// TwinCAT 3 PLC project ServerSampleProject
// ProgramVersion: 3.1.4026.23
// libraries:
//   Tc2_Standard, * (Beckhoff Automation GmbH)
//   Tc2_System, * (Beckhoff Automation GmbH)
//   Tc3_EventLogger, * (Beckhoff Automation GmbH)
//   Tc3_Module, * (Beckhoff Automation GmbH)
// project tree:
//   DUTs/Enums/ E_Enum_2.TcDUT, E_Operation.TcDUT, E_Enum_1.TcDUT
//   DUTs/Structures/ ST_Complex_1.TcDUT, ST_Complex_3.TcDUT, ST_Complex_4.TcDUT, ST_Complex_5.TcDUT, ST_Complex_6.TcDUT, ST_Complex_7.TcDUT, ST_Complex_8.TcDUT, ST_MathematicResults.TcDUT, ST_MathOperation.TcDUT, ST_Complex_2.TcDUT
//   GVLs/ GVL_alarm_condition.TcGVL, GVL_analog_items.TcGVL, GVL_historizing.TcGVL, GVL_inheritance.TcGVL, GVL_properties.TcGVL, Settings.TcGVL, GVL_enums.TcGVL, GVL_methods.TcGVL, GVL_structures.TcGVL, GVL_nodes_dynamic.TcGVL, GVL_nodes_static.TcGVL
//   / PlcTask.TcTTO
//   POUs/Inheritance/ FB_Base.TcPOU, FB_Derived.TcPOU
//   POUs/ MAIN.TcPOU
//   POUs/Methods/ FB_Job.TcPOU, FB_Mathematics.TcPOU, FB_Methods.TcPOU
//   POUs/Programs/ PRG_AlarmsConditions.TcPOU, PRG_Dynamic.TcPOU, PRG_Eventlogger.TcPOU, PRG_HistoricalAccess.TcPOU, PRG_Methods.TcPOU, PRG_Static.TcPOU
//   POUs/Properties/ FB_Properties.TcPOU
// real-time tasks:
//   TASK PlcTask: cycle T#10ms, priority 20, ADS port 350

CONFIGURATION ServerSampleProject
    RESOURCE PLC ON TwinCAT3
        TASK PlcTask(INTERVAL := T#10ms, PRIORITY := 20);
        PROGRAM MAIN WITH PlcTask : MAIN;
    END_RESOURCE
END_CONFIGURATION

// ---- DUTs/Enums/E_Enum_2.TcDUT
TYPE E_Enum_2 :
(
	ZERO := 0,
	ONE := 1,
	TWO := 2,
	THREE := 3,
	THIRTEEN := 13,
	the_answer_to_life_the_universe_and_everything := 42
) INT;
END_TYPE

// ---- DUTs/Enums/E_Operation.TcDUT
TYPE E_Operation :
(
	Addition := 0,
	Substract,
	Multiply,
	Divide
);
END_TYPE

// ---- DUTs/Enums/E_Enum_1.TcDUT
TYPE E_Enum_1 :
(
	ZERO := 0,
	ONE := 1,
	TWO := 2,
	THREE := 3,
	THIRTEEN := 13,
	the_answer_to_life_the_universe_and_everything := 42
);
END_TYPE

// ---- DUTs/Structures/ST_Complex_1.TcDUT
{attribute 'OPC.UA.DA' := '1'}
{attribute 'OPC.UA.DA.StructuredType' := '1'}
TYPE ST_Complex_1 :
STRUCT
	x 	: E_Enum_1;
	a 	: DINT;
	str : STRING;
	b 	: DINT;
END_STRUCT
END_TYPE

// ---- DUTs/Structures/ST_Complex_3.TcDUT
{attribute 'OPC.UA.DA' := '1'}
{attribute 'OPC.UA.DA.StructuredType' := '1'}
TYPE ST_Complex_3 :
STRUCT
	stAmsAddr : ST_AmsAddr;
END_STRUCT
END_TYPE

// ---- DUTs/Structures/ST_Complex_4.TcDUT
{attribute 'OPC.UA.DA' := '1'}
{attribute 'OPC.UA.DA.StructuredType' := '1'}
TYPE ST_Complex_4 :
STRUCT
	ErrorID : E_Enum_1;
END_STRUCT
END_TYPE

// ---- DUTs/Structures/ST_Complex_5.TcDUT
TYPE ST_Complex_5 :
STRUCT
	a : INT := 42;
	b : DINT := 43;
	c : REAL := 42.42;
	d : LREAL := 42.42;
	e : STRING := 'Hello TwinCAT';
	f : INT := 42;
	g : BOOL := TRUE;
END_STRUCT
END_TYPE

// ---- DUTs/Structures/ST_Complex_6.TcDUT
TYPE ST_Complex_6 :
STRUCT
	a : INT := 42;
	b : DINT := 43;
	c : REAL := 42.42;
	d : LREAL := 42.42;
	e : INT := 44;
	f : BOOL := TRUE;
END_STRUCT
END_TYPE

// ---- DUTs/Structures/ST_Complex_7.TcDUT
TYPE ST_Complex_7 :
STRUCT
	a : LREAL := 42.42;
	b : REAL := 42.42;
	c : REAL := 42.42;
END_STRUCT
END_TYPE

// ---- DUTs/Structures/ST_Complex_8.TcDUT
{attribute 'OPC.UA.DA' := '1'}
{attribute 'OPC.UA.DA.StructuredType' := '1'}
TYPE ST_Complex_8 :
STRUCT
	stComplex		: ST_Complex_1;
	strString5		: STRING[5]; (*String, max 5 chars*)
	eEnum	 		: E_Enum_1;
	strString3	 	: STRING[3]; (*String, max 3 chars*)
	arrComplex 		: ARRAY[0..1] OF ST_Complex_1;
	arrDint		 	: ARRAY[0..100] OF DINT;	
END_STRUCT
END_TYPE

// ---- DUTs/Structures/ST_MathematicResults.TcDUT
TYPE ST_MathematicResults :
STRUCT
	Sum : LREAL;
	Diff : LREAL;
	Prod : LREAL;
	Quo : LREAL;
END_STRUCT
END_TYPE

// ---- DUTs/Structures/ST_MathOperation.TcDUT
{attribute 'OPC.UA.DA.Description' := 'Structure to describe a math operation having one operator and two oparands'}
TYPE ST_MathOperation :
STRUCT
	operator : E_OPERATION; (*define the operator for calculation*)
	a : LREAL; (*First operand*)
	b : LREAL; (*Second operand*)
END_STRUCT
END_TYPE

// ---- DUTs/Structures/ST_Complex_2.TcDUT
{attribute 'OPC.UA.DA' := '1'}
{attribute 'OPC.UA.DA.StructuredType' := '1'}
TYPE ST_Complex_2 :
STRUCT
	c1 		: ST_Complex_1;
	s_5 	: STRING[5]; (*String, max 5 chars*)
	e 		: E_Enum_1;
	s_3 	: STRING[3]; (*String, max 3 chars*)
	cArr 	: ARRAY[0..5] OF ST_Complex_1;
	iArr 	: ARRAY[0..100] OF DINT;	
END_STRUCT
END_TYPE

// ---- GVLs/GVL_alarm_condition.TcGVL
VAR_GLOBAL
	{attribute 'OPC.UA.DA' := '1'}
	{attribute 'OPC.UA.DA.Description' := 'Triggers a LimitAlarmType when value reaches 10 or 0. Increments every 10 secs'}
	limitAlmTrigger: DINT;
	
	{attribute 'OPC.UA.DA' := '1'}
	{attribute 'OPC.UA.DA.Description' := 'Triggers an OffNormalAlarmType when set to true. State changes state every 10 secs.'}
	offNormAlmTrigger : BOOL;
END_VAR

// ---- GVLs/GVL_analog_items.TcGVL
{attribute 'qualified_only'}
VAR_GLOBAL
	{attribute 'OPC.UA.DA' := '1'}
	{attribute 'OPC.UA.DA.AnalogItemType' := '1'}
	{attribute 'OPC.UA.DA.AnalogItemType.EngineeringUnits' := '20529'  }(*EngeneeringUnit = percent*)
	{attribute 'OPC.UA.DA.AnalogItemType.InstrumentRange' := '0:100'  }
	{attribute 'OPC.UA.DA.AnalogItemType.EURange' := '10:90'  }
	{attribute 'OPC.UA.DA.AnalogItemType.WriteBehavior' := '1'  } (*AnalogWrMode_AllowAny = 0,
																	AnalogWrMode_Clamp = 1,
																	AnalogWrMode_Reject = 2,*)
	{attribute 'OPC.UA.DA.Description' := 'Analog item type. Write mode is clamped to instrument range'}
	analog_percent : REAL := 50;
	
	{attribute 'OPC.UA.DA' := '1'}
	{attribute 'OPC.UA.DA.AnalogItemType' := '1'}
	{attribute 'OPC.UA.DA.AnalogItemType.EngineeringUnits' := '12851'  }(*EngeneeringUnit = gram_per_cubic_centimetre*)
	{attribute 'OPC.UA.DA.AnalogItemType.InstrumentRange' := '0:100'  }
	{attribute 'OPC.UA.DA.AnalogItemType.EURange' := '0:75'  }
	{attribute 'OPC.UA.DA.AnalogItemType.WriteBehavior' := '2'  } (*AnalogWrMode_AllowAny = 0,
																	AnalogWrMode_Clamp = 1,
																	AnalogWrMode_Reject = 2,*)
	{attribute 'OPC.UA.DA.Description' := 'Analog item type. Write is rejected when out of instrument range'}
	analog_gram_per_cubic_centimetre : REAL := 50;	
	
	{attribute 'OPC.UA.DA' := '1'}
	{attribute 'OPC.UA.DA.AnalogItemType' := '1'}
	{attribute 'OPC.UA.DA.AnalogItemType.EngineeringUnits' := '5257525'  }(*EngeneeringUnit = megabyte_per_second*)
	{attribute 'OPC.UA.DA.AnalogItemType.EURange' := '0:10'  }
	{attribute 'OPC.UA.DA.AnalogItemType.InstrumentRange' := '0:100'  }
	{attribute 'OPC.UA.DA.AnalogItemType.WriteBehavior' := '0'  } (*AnalogWrMode_AllowAny = 0,
																	AnalogWrMode_Clamp = 1,
																	AnalogWrMode_Reject = 2,*)
	{attribute 'OPC.UA.DA.Description' := 'Analog item type. Write mode allows writing out of Instrument range'}
	analog_mbps : REAL;	
	
	{attribute 'OPC.UA.DA' := '1'}
	{attribute 'OPC.UA.DA.AnalogItemType' := '1'}
	{attribute 'OPC.UA.DA.AnalogItemType.EngineeringUnits' := '20529'  }(*EngeneeringUnit = percent*)
	{attribute 'OPC.UA.DA.AnalogItemType.InstrumentRange' := '0:100'  }
	{attribute 'OPC.UA.DA.AnalogItemType.EURange' := '10:90'  }
	{attribute 'OPC.UA.DA.AnalogItemType.WriteBehavior' := '2'  } (*AnalogWrMode_AllowAny = 0,
																	AnalogWrMode_Clamp = 1,
																	AnalogWrMode_Reject = 2,*)
	{attribute 'OPC.UA.DA.Description' := 'Analog item of type Double. '}
	analog_dbl : LREAL := 50;	
	
	{attribute 'OPC.UA.DA' := '1'}
	{attribute 'OPC.UA.DA.AnalogItemType' := '1'}
	{attribute 'OPC.UA.DA.AnalogItemType.EngineeringUnits' := '20529'  }(*EngeneeringUnit = percent*)
	{attribute 'OPC.UA.DA.AnalogItemType.InstrumentRange' := '0:100'  }
	{attribute 'OPC.UA.DA.AnalogItemType.EURange' := '10:90'  }
	{attribute 'OPC.UA.DA.AnalogItemType.WriteBehavior' := '2'  } (*AnalogWrMode_AllowAny = 0,
																	AnalogWrMode_Clamp = 1,
																	AnalogWrMode_Reject = 2,*)
	{attribute 'OPC.UA.DA.Description' := 'Analog item of type Float. '}
	analog_flt : REAL := 50;		
	
	{attribute 'OPC.UA.DA' := '1'}
	{attribute 'OPC.UA.DA.AnalogItemType' := '1'}
	{attribute 'OPC.UA.DA.AnalogItemType.EngineeringUnits' := '20529'  }(*EngeneeringUnit = percent*)
	{attribute 'OPC.UA.DA.AnalogItemType.InstrumentRange' := '0:100'  }
	{attribute 'OPC.UA.DA.AnalogItemType.EURange' := '10:90'  }
	{attribute 'OPC.UA.DA.AnalogItemType.WriteBehavior' := '2'  } (*AnalogWrMode_AllowAny = 0,
																	AnalogWrMode_Clamp = 1,
																	AnalogWrMode_Reject = 2,*)
	{attribute 'OPC.UA.DA.Description' := 'Analog item of type Int16. '}
	analog_i16 : INT := 50;		
	
	{attribute 'OPC.UA.DA' := '1'}
	{attribute 'OPC.UA.DA.AnalogItemType' := '1'}
	{attribute 'OPC.UA.DA.AnalogItemType.EngineeringUnits' := '20529'  }(*EngeneeringUnit = percent*)
	{attribute 'OPC.UA.DA.AnalogItemType.InstrumentRange' := '0:100'  }
	{attribute 'OPC.UA.DA.AnalogItemType.EURange' := '10:90'  }
	{attribute 'OPC.UA.DA.AnalogItemType.WriteBehavior' := '2'  } (*AnalogWrMode_AllowAny = 0,
																	AnalogWrMode_Clamp = 1,
																	AnalogWrMode_Reject = 2,*)
	{attribute 'OPC.UA.DA.Description' := 'Analog item of type UInt16. '}
	analog_ui16 : UINT := 50;		
	
	{attribute 'OPC.UA.DA' := '1'}
	{attribute 'OPC.UA.DA.AnalogItemType' := '1'}
	{attribute 'OPC.UA.DA.AnalogItemType.EngineeringUnits' := '20529'  }(*EngeneeringUnit = percent*)
	{attribute 'OPC.UA.DA.AnalogItemType.InstrumentRange' := '0:100'  }
	{attribute 'OPC.UA.DA.AnalogItemType.EURange' := '10:90'  }
	{attribute 'OPC.UA.DA.AnalogItemType.WriteBehavior' := '2'  } (*AnalogWrMode_AllowAny = 0,
																	AnalogWrMode_Clamp = 1,
																	AnalogWrMode_Reject = 2,*)
	{attribute 'OPC.UA.DA.Description' := 'Analog item of type Int32. '}
	analog_i32 : DINT := 50;		

	{attribute 'OPC.UA.DA' := '1'}
	{attribute 'OPC.UA.DA.AnalogItemType' := '1'}
	{attribute 'OPC.UA.DA.AnalogItemType.EngineeringUnits' := '20529'  }(*EngeneeringUnit = percent*)
	{attribute 'OPC.UA.DA.AnalogItemType.InstrumentRange' := '0:100'  }
	{attribute 'OPC.UA.DA.AnalogItemType.EURange' := '10:90'  }
	{attribute 'OPC.UA.DA.AnalogItemType.WriteBehavior' := '2'  } (*AnalogWrMode_AllowAny = 0,
																	AnalogWrMode_Clamp = 1,
																	AnalogWrMode_Reject = 2,*)
	{attribute 'OPC.UA.DA.Description' := 'Analog item of type UInt32. '}
	analog_ui32 : UDINT := 50;
	
	{attribute 'OPC.UA.DA' := '1'}
	{attribute 'OPC.UA.DA.AnalogItemType' := '1'}
	{attribute 'OPC.UA.DA.AnalogItemType.EngineeringUnits' := '20529'  }(*EngeneeringUnit = percent*)
	{attribute 'OPC.UA.DA.AnalogItemType.InstrumentRange' := '0:100'  }
	{attribute 'OPC.UA.DA.AnalogItemType.EURange' := '10:90'  }
	{attribute 'OPC.UA.DA.AnalogItemType.WriteBehavior' := '2'  } (*AnalogWrMode_AllowAny = 0,
																	AnalogWrMode_Clamp = 1,
																	AnalogWrMode_Reject = 2,*)
	{attribute 'OPC.UA.DA.Description' := 'Analog item of type Int64. '}
	analog_i64 : LINT := 50;		
	
	{attribute 'OPC.UA.DA' := '1'}
	{attribute 'OPC.UA.DA.AnalogItemType' := '1'}
	{attribute 'OPC.UA.DA.AnalogItemType.EngineeringUnits' := '20529'  }(*EngeneeringUnit = percent*)
	{attribute 'OPC.UA.DA.AnalogItemType.InstrumentRange' := '0:100'  }
	{attribute 'OPC.UA.DA.AnalogItemType.EURange' := '10:90'  }
	{attribute 'OPC.UA.DA.AnalogItemType.WriteBehavior' := '2'  } (*AnalogWrMode_AllowAny = 0,
																	AnalogWrMode_Clamp = 1,
																	AnalogWrMode_Reject = 2,*)
	{attribute 'OPC.UA.DA.Description' := 'Analog item of type UInt64. '}
	analog_ui64 : ULINT := 50;		
	
	{attribute 'OPC.UA.DA' := '1'}
	{attribute 'OPC.UA.DA.AnalogItemType' := '1'}
	{attribute 'OPC.UA.DA.AnalogItemType.EngineeringUnits' := '20529'  }(*EngeneeringUnit = percent*)
	{attribute 'OPC.UA.DA.AnalogItemType.InstrumentRange' := '0:100'  }
	{attribute 'OPC.UA.DA.AnalogItemType.EURange' := '10:90'  }
	{attribute 'OPC.UA.DA.AnalogItemType.WriteBehavior' := '2'  } (*AnalogWrMode_AllowAny = 0,
																	AnalogWrMode_Clamp = 1,
																	AnalogWrMode_Reject = 2,*)
	{attribute 'OPC.UA.DA.Description' := 'Analog item of type SByte. '}
	analog_i8 : SINT := 50;		
	
	{attribute 'OPC.UA.DA' := '1'}
	{attribute 'OPC.UA.DA.AnalogItemType' := '1'}
	{attribute 'OPC.UA.DA.AnalogItemType.EngineeringUnits' := '20529'  }(*EngeneeringUnit = percent*)
	{attribute 'OPC.UA.DA.AnalogItemType.InstrumentRange' := '0:100'  }
	{attribute 'OPC.UA.DA.AnalogItemType.EURange' := '10:90'  }
	{attribute 'OPC.UA.DA.AnalogItemType.WriteBehavior' := '2'  } (*AnalogWrMode_AllowAny = 0,
																	AnalogWrMode_Clamp = 1,
																	AnalogWrMode_Reject = 2,*)
	{attribute 'OPC.UA.DA.Description' := 'Analog item of type Byte. '}
	analog_ui8 : USINT := 50;	
END_VAR

// ---- GVLs/GVL_historizing.TcGVL
VAR_GLOBAL
	
	{attribute 'OPC.UA.DA' := '1'}
	{attribute 'OPC.UA.DA.Description' := 'HistoricalAccess with Volatile storage'}
	volatile_sinus	: LREAL;
	{attribute 'OPC.UA.DA' := '1'}
	{attribute 'OPC.UA.DA.Description' := 'HistoricalAccess with Volatile storage'}	
	volatile_cosinus : LREAL;
	{attribute 'OPC.UA.DA' := '1'}
	{attribute 'OPC.UA.DA.Description' := 'HistoricalAccess with Volatile storage'}	
	volatile_cosinushalf : LREAL;
	{attribute 'OPC.UA.DA' := '1'}
	{attribute 'OPC.UA.DA.Description' := 'HistoricalAccess with SQLite storage'}
	sqlite_sinus : LREAL;
	{attribute 'OPC.UA.DA' := '1'}
	{attribute 'OPC.UA.DA.Description' := 'HistoricalAccess with SQLite storage'}	
	sqlite_cosinus : LREAL;
	{attribute 'OPC.UA.DA' := '1'}
	{attribute 'OPC.UA.DA.Description' := 'HistoricalAccess with SQLite storage'}	
	sqlite_cosinushalf : LREAL;

END_VAR

// ---- GVLs/GVL_inheritance.TcGVL
{attribute 'qualified_only'}
VAR_GLOBAL
	{attribute 'OPC.UA.DA' := '1'}
	{attribute 'OPC.UA.DA.Description' := 'Base class'}
	BaseType : FB_Base;
	
	{attribute 'OPC.UA.DA' := '1'}
	{attribute 'OPC.UA.DA.Description' := 'Derived class'}
	DerivedType : FB_Derived;	
END_VAR

// ---- GVLs/GVL_properties.TcGVL
{attribute 'qualified_only'}
VAR_GLOBAL
	{attribute 'OPC.UA.DA' := '1'}
	Properties : FB_Properties;
END_VAR

// ---- GVLs/Settings.TcGVL
VAR_GLOBAL
	{attribute 'OPC.UA.DA' := '1'}
	{attribute 'OPC.UA.DA.Description' := 'Sets PLC update interval of variables in GVL_nodes_dynamic'} 	
	UpdateTimer : TON := (PT:=T#10MS);
END_VAR
VAR_GLOBAL CONSTANT
	ARRSIZEX : INT := 10; 
	ARRSIZEY : INT := 10; 
	ARRSIZEZ : INT := 10;
	ARRSIZEHUGE : INT := 10000;
END_VAR

// ---- GVLs/GVL_enums.TcGVL
{attribute 'qualified_only'}
VAR_GLOBAL
	{attribute 'OPC.UA.DA' := '1'}
	{attribute 'OPC.UA.DA.Description' := 'Enumeration type (DINT)'} 
	Enum1 : E_Enum_1;
	{attribute 'OPC.UA.DA' := '1'}
	{attribute 'OPC.UA.DA.Description' := 'Enumeration type (INT)'} 
	Enum2 : E_Enum_2;	
END_VAR

// ---- GVLs/GVL_methods.TcGVL
VAR_GLOBAL
	{attribute 'OPC.UA.DA' := '1'}
	{attribute 'OPC.UA.DA.Description' := 'Methods with different InputOutput types'} 	
	Methods : FB_Methods;
	
	{attribute 'OPC.UA.DA' := '1'}
	{attribute 'OPC.UA.DA.Description' := 'Methods with mathematical functions'}
	Mathematics : FB_Mathematics;

	{attribute 'OPC.UA.DA' := '1'}
	{attribute 'OPC.UA.DA.Description' := 'Job method which execution may take longer than a PLC cycle'}
	Job : FB_Job;	
END_VAR

// ---- GVLs/GVL_structures.TcGVL
VAR_GLOBAL
	{attribute 'OPC.UA.DA' := '1'}
	{attribute 'OPC.UA.DA.StructuredType' := '1'}
	{attribute 'OPC.UA.DA.Description' := 'Complex (structured) type '} 	
	StructuredType1 : ST_Complex_1;
	
	{attribute 'OPC.UA.DA' := '2'}
	{attribute 'OPC.UA.DA.StructuredType' := '1'}
	{attribute 'OPC.UA.DA.Description' := 'Complex (structured) type '} 	
	StructuredType1WithoutMember : ST_Complex_1;

	{attribute 'OPC.UA.DA' := '1'}
	{attribute 'OPC.UA.DA.StructuredType' := '1'}
	{attribute 'OPC.UA.DA.Description' := 'Complex (structured) type '} 		
	StructuredType2 : ST_Complex_2;
	
	{attribute 'OPC.UA.DA' := '1'}
	{attribute 'OPC.UA.DA.StructuredType' := '1'}
	{attribute 'OPC.UA.DA.Description' := 'Complex (structured) type '} 		
	StructuredType3 : ST_Complex_3;

	{attribute 'OPC.UA.DA' := '1'}
	{attribute 'OPC.UA.DA.StructuredType' := '1'}
	{attribute 'OPC.UA.DA.Description' := 'Complex (structured) type '} 		
	StructuredType4 : ST_Complex_4;	
	
	{attribute 'OPC.UA.DA' := '1'}
	{attribute 'OPC.UA.DA.StructuredType' := '1'}
	{attribute 'OPC.UA.DA.Description' := 'Complex (structured) type '} 		
	StructuredType5 : ST_Complex_5;	
	
	{attribute 'OPC.UA.DA' := '1'}
	{attribute 'OPC.UA.DA.StructuredType' := '1'}
	{attribute 'OPC.UA.DA.Description' := 'Complex (structured) type '} 		
	StructuredType6 : ST_Complex_6;	
	
	{attribute 'OPC.UA.DA' := '1'}
	{attribute 'OPC.UA.DA.StructuredType' := '1'}
	{attribute 'OPC.UA.DA.Description' := 'Complex (structured) type '} 		
	StructuredType7 : ST_Complex_7;		

	{attribute 'OPC.UA.DA' := '1'}
	{attribute 'OPC.UA.DA.StructuredType' := '1'}
	{attribute 'OPC.UA.DA.Description' := 'Complex (structured) type '} 		
	StructuredType8 : ST_Complex_8;	
	
	{attribute 'OPC.UA.DA' := '1'}
	{attribute 'OPC.UA.DA.StructuredType' := '1'}
	{attribute 'OPC.UA.DA.Description' := 'Array of complex (structured) type'} 	
	arrStComplex : ARRAY[0..ARRSIZEX] OF ST_Complex_1;

	{attribute 'OPC.UA.DA' := '1'}
	{attribute 'OPC.UA.DA.StructuredType' := '1'}
	{attribute 'OPC.UA.DA.Description' := 'Array of complex (structured) type'} 		
	arrStComplex2 : ARRAY[0..ARRSIZEX] OF ST_Complex_2;		
END_VAR

// ---- GVLs/GVL_nodes_dynamic.TcGVL
VAR_GLOBAL
	//scalars
	{attribute 'OPC.UA.DA' := '1'}
	{attribute 'OPC.UA.DA.Description' := 'Scalar BOOL, modified by a TRIG'}	
	dyn_scalar_BOOL_trigger : BOOL;
	{attribute 'OPC.UA.DA' := '1'}
	{attribute 'OPC.UA.DA.Description' := 'Scalar BOOL'} 
	dyn_scalar_BOOL	: BOOL;(* ~ 	(OPC : 1 : available for OPC-clients) *)
	{attribute 'OPC.UA.DA' := '1'}
	{attribute 'OPC.UA.DA.Description' := 'Scalar SINT'}
	dyn_scalar_I1	: SINT;		(* ~ 	(OPC : 1 : available for OPC-clients) *)					
	{attribute 'OPC.UA.DA' := '1'}
	{attribute 'OPC.UA.DA.Description' := 'Scalar USINT'}	
	dyn_scalar_UI1	: USINT;	(* ~ 	(OPC : 1 : available for OPC-clients) *)					
	{attribute 'OPC.UA.DA' := '1'}
	{attribute 'OPC.UA.DA.Description' := 'Scalar INT'}	
	dyn_scalar_I2 	: INT;			(* ~ 	(OPC : 1 : available for OPC-clients) *)				
	{attribute 'OPC.UA.DA' := '1'}
	{attribute 'OPC.UA.DA.Description' := 'Scalar UINT'}	
	dyn_scalar_UI2	: UINT;			(* ~ 	(OPC : 1 : available for OPC-clients) *)				
	{attribute 'OPC.UA.DA' := '1'}
	{attribute 'OPC.UA.DA.Description' := 'Scalar DINT'}	
	dyn_scalar_I4	: DINT;		(* ~ 	(OPC : 1 : available for OPC-clients) *)					
	{attribute 'OPC.UA.DA' := '1'}
	{attribute 'OPC.UA.DA.Description' := 'Scalar UDINT'}	
	dyn_scalar_UI4	: UDINT;(* ~ 	(OPC : 1 : available for OPC-clients) *)
	{attribute 'OPC.UA.DA' := '1'}
	{attribute 'OPC.UA.DA.Description' := 'Scalar LINT'}
	dyn_scalar_I8	: LINT;	(* ~ 	(OPC : 1 : available for OPC-clients) *)
	{attribute 'OPC.UA.DA' := '1'}
	{attribute 'OPC.UA.DA.Description' := 'Scalar ULINT'}
	dyn_scalar_UI8	: ULINT;(* ~ 	(OPC : 1 : available for OPC-clients) *)
	{attribute 'OPC.UA.DA' := '1'}
	{attribute 'OPC.UA.DA.Description' := 'Scalar BYTE'}
	dyn_scalar_BYTE	: BYTE;(* ~ 	(OPC : 1 : available for OPC-clients) *)
	{attribute 'OPC.UA.DA' := '1'}
	{attribute 'OPC.UA.DA.Description' := 'Scalar WORD'}	
	dyn_scalar_WORD	: WORD;(* ~ 	(OPC : 1 : available for OPC-clients) *)
	{attribute 'OPC.UA.DA' := '1'}
	{attribute 'OPC.UA.DA.Description' := 'Scalar DWORD'}	
	dyn_scalar_DWORD: DWORD;(* ~ 	(OPC : 1 : available for OPC-clients) *)
	{attribute 'OPC.UA.DA' := '1'}
	{attribute 'OPC.UA.DA.Description' := 'Scalar LWORD'}	
	dyn_scalar_LWORD: LWORD;(* ~ 	(OPC : 1 : available for OPC-clients) *)
	{attribute 'OPC.UA.DA' := '1'}
	{attribute 'OPC.UA.DA.Description' := 'Scalar REAL'}	
	dyn_scalar_R4	: REAL;(* ~ 	(OPC : 1 : available for OPC-clients) *)
	{attribute 'OPC.UA.DA' := '1'}
	{attribute 'OPC.UA.DA.Description' := 'Scalar LREAL'}
	dyn_scalar_R8	: LREAL;(* ~ 	(OPC : 1 : available for OPC-clients) *)
	{attribute 'OPC.UA.DA' := '1'}
	{attribute 'OPC.UA.DA.Description' := 'Scalar STRING'}	
	dyn_scalar_BSTR	: STRING;(* ~ 	(OPC : 1 : available for OPC-clients) *)
	{attribute 'OPC.UA.DA' := '1'}
	{attribute 'OPC.UA.DA.Description' := 'Scalar CHAR'}	
	//dyn_scalar_CHAR	: CHAR;
	{attribute 'OPC.UA.DA' := '1'}
	{attribute 'OPC.UA.DA.Description' := 'Scalar WSTRING'}	
	dyn_scalar_WSTRING : WSTRING;(* ~ 	(OPC : 1 : available for OPC-clients) *)
	{attribute 'OPC.UA.DA' := '1'}
	{attribute 'OPC.UA.DA.Description' := 'Scalar WCHAR'}	
	//dyn_scalar_WCHAR: WCHAR;
	{attribute 'OPC.UA.DA' := '1'}
	{attribute 'OPC.UA.DA.Description' := 'Scalar DT'}	
	dyn_scalar_DT	: DT;(* ~ 	(OPC : 1 : available for OPC-clients) *)
	{attribute 'OPC.UA.DA' := '1'}
	{attribute 'OPC.UA.DA.Description' := 'Scalar DATE'}	
	dyn_scalar_DATE : DATE;(* ~ 	(OPC : 1 : available for OPC-clients) *)
	{attribute 'OPC.UA.DA' := '1'}
	{attribute 'OPC.UA.DA.Description' := 'Scalar TOD'}	
	dyn_scalar_TOD	: TOD;(* ~ 	(OPC : 1 : available for OPC-clients) *)
	{attribute 'OPC.UA.DA' := '1'}
	{attribute 'OPC.UA.DA.Description' := 'Scalar TIME'}	
	dyn_scalar_TIME	: TIME;(* ~ 	(OPC : 1 : available for OPC-clients) *)
	
	//1dim
	{attribute 'OPC.UA.DA' := '1'}
	{attribute 'OPC.UA.DA.Description' := '1dim Array BOOL'}	
	dyn_1dim_BOOL	: ARRAY[0..ARRSIZEX] OF BOOL;(* ~ 	(OPC : 1 : available for OPC-clients) *)
	{attribute 'OPC.UA.DA' := '1'}
	{attribute 'OPC.UA.DA.Description' := '1dim Array BOOL'}	
	dyn_1dim_I1		: ARRAY[0..ARRSIZEX] OF SINT;(* ~ 	(OPC : 1 : available for OPC-clients) *)
	{attribute 'OPC.UA.DA' := '1'}
	{attribute 'OPC.UA.DA.Description' := '1dim Array BOOL'}	
	dyn_1dim_I1_Huge: ARRAY[0..ARRSIZEHUGE] OF SINT;(* ~ 	(OPC : 1 : available for OPC-clients) *)	
	{attribute 'OPC.UA.DA' := '1'}
	{attribute 'OPC.UA.DA.Description' := '1dim Array BOOL'}
	dyn_1dim_UI1	: ARRAY[0..ARRSIZEX] OF USINT;(* ~ 	(OPC : 1 : available for OPC-clients) *)
	{attribute 'OPC.UA.DA' := '1'}
	{attribute 'OPC.UA.DA.Description' := '1dim Array BOOL'}
	dyn_1dim_I2 	: ARRAY[0..ARRSIZEX] OF INT;(* ~ 	(OPC : 1 : available for OPC-clients) *)
	{attribute 'OPC.UA.DA' := '1'}
	{attribute 'OPC.UA.DA.Description' := '1dim Array BOOL'}	
	dyn_1dim_UI2	: ARRAY[0..ARRSIZEX] OF UINT;(* ~ 	(OPC : 1 : available for OPC-clients) *)
	{attribute 'OPC.UA.DA' := '1'}
	{attribute 'OPC.UA.DA.Description' := '1dim Array BOOL'}	
	dyn_1dim_I4		: ARRAY[0..ARRSIZEX] OF DINT;(* ~ 	(OPC : 1 : available for OPC-clients) *)
	{attribute 'OPC.UA.DA' := '1'}
	{attribute 'OPC.UA.DA.Description' := '1dim Array BOOL'}	
	dyn_1dim_I4_Huge: ARRAY[0..ARRSIZEHUGE] OF DINT;(* ~ 	(OPC : 1 : available for OPC-clients) *)	
	{attribute 'OPC.UA.DA' := '1'}
	{attribute 'OPC.UA.DA.Description' := '1dim Array BOOL'}
	dyn_1dim_UI4	: ARRAY[0..ARRSIZEX] OF UDINT;(* ~ 	(OPC : 1 : available for OPC-clients) *)
	{attribute 'OPC.UA.DA' := '1'}
	{attribute 'OPC.UA.DA.Description' := '1dim Array BOOL'}
	dyn_1dim_I8		: ARRAY[0..ARRSIZEX] OF LINT;(* ~ 	(OPC : 1 : available for OPC-clients) *)
	{attribute 'OPC.UA.DA' := '1'}
	{attribute 'OPC.UA.DA.Description' := '1dim Array BOOL'}
	dyn_1dim_UI8	: ARRAY[0..ARRSIZEX] OF ULINT;(* ~ 	(OPC : 1 : available for OPC-clients) *)
	{attribute 'OPC.UA.DA' := '1'}
	{attribute 'OPC.UA.DA.Description' := '1dim Array BOOL'}
	dyn_1dim_BYTE	: ARRAY[0..ARRSIZEX] OF BYTE;(* ~ 	(OPC : 1 : available for OPC-clients) *)
	{attribute 'OPC.UA.DA' := '1'}
	{attribute 'OPC.UA.DA.Description' := '1dim Array BOOL'}
	dyn_1dim_WORD	: ARRAY[0..ARRSIZEX] OF WORD;(* ~ 	(OPC : 1 : available for OPC-clients) *)
	{attribute 'OPC.UA.DA' := '1'}
	{attribute 'OPC.UA.DA.Description' := '1dim Array BOOL'}
	dyn_1dim_DWORD	: ARRAY[0..ARRSIZEX] OF DWORD;(* ~ 	(OPC : 1 : available for OPC-clients) *)
	{attribute 'OPC.UA.DA' := '1'}
	{attribute 'OPC.UA.DA.Description' := '1dim Array BOOL'}
	dyn_1dim_LWORD	: ARRAY[0..ARRSIZEX] OF LWORD;(* ~ 	(OPC : 1 : available for OPC-clients) *)
	{attribute 'OPC.UA.DA' := '1'}
	{attribute 'OPC.UA.DA.Description' := '1dim Array BOOL'}
	dyn_1dim_R4		: ARRAY[0..ARRSIZEX] OF REAL;(* ~ 	(OPC : 1 : available for OPC-clients) *)
	{attribute 'OPC.UA.DA' := '1'}
	{attribute 'OPC.UA.DA.Description' := '1dim Array BOOL'}
	dyn_1dim_R8		: ARRAY[0..ARRSIZEX] OF LREAL;(* ~ 	(OPC : 1 : available for OPC-clients) *)
	{attribute 'OPC.UA.DA' := '1'}
	{attribute 'OPC.UA.DA.Description' := '1dim Array BOOL'}
	dyn_1dim_BSTR	: ARRAY[0..ARRSIZEX] OF STRING;(* ~ 	(OPC : 1 : available for OPC-clients) *)
	{attribute 'OPC.UA.DA' := '1'}
	{attribute 'OPC.UA.DA.Description' := '1dim Array BOOL'}
	//dyn_1dim_CHAR	: ARRAY[0..ARRSIZEX] OF CHAR;
	{attribute 'OPC.UA.DA' := '1'}
	{attribute 'OPC.UA.DA.Description' := '1dim Array BOOL'}
	dyn_1dim_WSTRING : ARRAY[0..ARRSIZEX] OF WSTRING;(* ~ 	(OPC : 1 : available for OPC-clients) *)
	{attribute 'OPC.UA.DA' := '1'}
	{attribute 'OPC.UA.DA.Description' := '1dim Array BOOL'}
	//dyn_1dim_WCHAR: ARRAY[0..ARRSIZEX] OF WCHAR;
	{attribute 'OPC.UA.DA' := '1'}
	{attribute 'OPC.UA.DA.Description' := '1dim Array BOOL'}
	dyn_1dim_DT		: ARRAY[0..ARRSIZEX] OF DT;(* ~ 	(OPC : 1 : available for OPC-clients) *)
	{attribute 'OPC.UA.DA' := '1'}
	{attribute 'OPC.UA.DA.Description' := '1dim Array BOOL'}
	dyn_1dim_DATE 	: ARRAY[0..ARRSIZEX] OF DATE;(* ~ 	(OPC : 1 : available for OPC-clients) *)
	{attribute 'OPC.UA.DA' := '1'}
	{attribute 'OPC.UA.DA.Description' := '1dim Array BOOL'}
	dyn_1dim_TOD	: ARRAY[0..ARRSIZEX] OF TOD;(* ~ 	(OPC : 1 : available for OPC-clients) *)
	{attribute 'OPC.UA.DA' := '1'}
	{attribute 'OPC.UA.DA.Description' := '1dim Array BOOL'}
	dyn_1dim_TIME	: ARRAY[0..ARRSIZEX] OF TIME;(* ~ 	(OPC : 1 : available for OPC-clients) *)
	
	//2dim
	{attribute 'OPC.UA.DA' := '1'}
	{attribute 'OPC.UA.DA.Description' := '2dim Array BOOL'}
	dyn_2dim_BOOL	: ARRAY[0..ARRSIZEX, 0..ARRSIZEY] OF BOOL;(* ~ 	(OPC : 1 : available for OPC-clients) *)
	{attribute 'OPC.UA.DA' := '1'}
	{attribute 'OPC.UA.DA.Description' := '2dim Array BOOL'}
	dyn_2dim_I1		: ARRAY[0..ARRSIZEX, 0..ARRSIZEY] OF SINT;(* ~ 	(OPC : 1 : available for OPC-clients) *)
	{attribute 'OPC.UA.DA' := '1'}
	{attribute 'OPC.UA.DA.Description' := '2dim Array BOOL'}
	dyn_2dim_UI1	: ARRAY[0..ARRSIZEX, 0..ARRSIZEY] OF USINT;(* ~ 	(OPC : 1 : available for OPC-clients) *)
	{attribute 'OPC.UA.DA' := '1'}
	{attribute 'OPC.UA.DA.Description' := '2dim Array BOOL'}
	dyn_2dim_I2 	: ARRAY[0..ARRSIZEX, 0..ARRSIZEY] OF INT;(* ~ 	(OPC : 1 : available for OPC-clients) *)
	{attribute 'OPC.UA.DA' := '1'}
	{attribute 'OPC.UA.DA.Description' := '2dim Array BOOL'}
	dyn_2dim_UI2	: ARRAY[0..ARRSIZEX, 0..ARRSIZEY] OF UINT;(* ~ 	(OPC : 1 : available for OPC-clients) *)
	{attribute 'OPC.UA.DA' := '1'}
	{attribute 'OPC.UA.DA.Description' := '2dim Array BOOL'}
	dyn_2dim_I4		: ARRAY[0..ARRSIZEX, 0..ARRSIZEY] OF DINT;(* ~ 	(OPC : 1 : available for OPC-clients) *)
	{attribute 'OPC.UA.DA' := '1'}
	{attribute 'OPC.UA.DA.Description' := '2dim Array BOOL'}
	dyn_2dim_UI4	: ARRAY[0..ARRSIZEX, 0..ARRSIZEY] OF UDINT;(* ~ 	(OPC : 1 : available for OPC-clients) *)
	{attribute 'OPC.UA.DA' := '1'}
	{attribute 'OPC.UA.DA.Description' := '2dim Array BOOL'}
	dyn_2dim_I8		: ARRAY[0..ARRSIZEX, 0..ARRSIZEY] OF LINT;(* ~ 	(OPC : 1 : available for OPC-clients) *)
	{attribute 'OPC.UA.DA' := '1'}
	{attribute 'OPC.UA.DA.Description' := '2dim Array BOOL'}
	dyn_2dim_UI8	: ARRAY[0..ARRSIZEX, 0..ARRSIZEY] OF ULINT;(* ~ 	(OPC : 1 : available for OPC-clients) *)
	{attribute 'OPC.UA.DA' := '1'}
	{attribute 'OPC.UA.DA.Description' := '2dim Array BOOL'}
	dyn_2dim_BYTE	: ARRAY[0..ARRSIZEX, 0..ARRSIZEY] OF BYTE;(* ~ 	(OPC : 1 : available for OPC-clients) *)
	{attribute 'OPC.UA.DA' := '1'}
	{attribute 'OPC.UA.DA.Description' := '2dim Array BOOL'}
	dyn_2dim_WORD	: ARRAY[0..ARRSIZEX, 0..ARRSIZEY] OF WORD;(* ~ 	(OPC : 1 : available for OPC-clients) *)
	{attribute 'OPC.UA.DA' := '1'}
	{attribute 'OPC.UA.DA.Description' := '2dim Array BOOL'}
	dyn_2dim_DWORD	: ARRAY[0..ARRSIZEX, 0..ARRSIZEY] OF DWORD;(* ~ 	(OPC : 1 : available for OPC-clients) *)
	{attribute 'OPC.UA.DA' := '1'}
	{attribute 'OPC.UA.DA.Description' := '2dim Array BOOL'}
	dyn_2dim_LWORD	: ARRAY[0..ARRSIZEX, 0..ARRSIZEY] OF LWORD;(* ~ 	(OPC : 1 : available for OPC-clients) *)
	{attribute 'OPC.UA.DA' := '1'}
	{attribute 'OPC.UA.DA.Description' := '2dim Array BOOL'}
	dyn_2dim_R4		: ARRAY[0..ARRSIZEX, 0..ARRSIZEY] OF REAL;(* ~ 	(OPC : 1 : available for OPC-clients) *)
	{attribute 'OPC.UA.DA' := '1'}
	{attribute 'OPC.UA.DA.Description' := '2dim Array BOOL'}
	dyn_2dim_R8		: ARRAY[0..ARRSIZEX, 0..ARRSIZEY] OF LREAL;(* ~ 	(OPC : 1 : available for OPC-clients) *)
	{attribute 'OPC.UA.DA' := '1'}
	{attribute 'OPC.UA.DA.Description' := '2dim Array BOOL'}
	dyn_2dim_BSTR	: ARRAY[0..ARRSIZEX, 0..ARRSIZEY] OF STRING;(* ~ 	(OPC : 1 : available for OPC-clients) *)
	{attribute 'OPC.UA.DA' := '1'}
	{attribute 'OPC.UA.DA.Description' := '2dim Array BOOL'}
	//dyn_2dim_CHAR	: ARRAY[0..ARRSIZEX, 0..ARRSIZEY] OF CHAR;
	{attribute 'OPC.UA.DA' := '1'}
	{attribute 'OPC.UA.DA.Description' := '2dim Array BOOL'}
	dyn_2dim_WSTRING : ARRAY[0..ARRSIZEX, 0..ARRSIZEY] OF WSTRING;(* ~ 	(OPC : 1 : available for OPC-clients) *)
	{attribute 'OPC.UA.DA' := '1'}
	{attribute 'OPC.UA.DA.Description' := '2dim Array BOOL'}
	//dyn_2dim_WCHAR: ARRAY[0..ARRSIZEX, 0..ARRSIZEY] OF WCHAR;
	{attribute 'OPC.UA.DA' := '1'}
	{attribute 'OPC.UA.DA.Description' := '2dim Array BOOL'}
	dyn_2dim_DT		: ARRAY[0..ARRSIZEX, 0..ARRSIZEY] OF DT;(* ~ 	(OPC : 1 : available for OPC-clients) *)
	{attribute 'OPC.UA.DA' := '1'}
	{attribute 'OPC.UA.DA.Description' := '2dim Array BOOL'}
	dyn_2dim_DATE 	: ARRAY[0..ARRSIZEX, 0..ARRSIZEY] OF DATE;(* ~ 	(OPC : 1 : available for OPC-clients) *)
	{attribute 'OPC.UA.DA' := '1'}
	{attribute 'OPC.UA.DA.Description' := '2dim Array BOOL'}
	dyn_2dim_TOD	: ARRAY[0..ARRSIZEX, 0..ARRSIZEY] OF TOD;(* ~ 	(OPC : 1 : available for OPC-clients) *)
	{attribute 'OPC.UA.DA' := '1'}
	{attribute 'OPC.UA.DA.Description' := '2dim Array BOOL'}
	dyn_2dim_TIME	: ARRAY[0..ARRSIZEX, 0..ARRSIZEY] OF TIME;(* ~ 	(OPC : 1 : available for OPC-clients) *)

	//3dim
	{attribute 'OPC.UA.DA' := '1'}
	{attribute 'OPC.UA.DA.Description' := '3dim Array BOOL'}
	dyn_3dim_BOOL	: ARRAY[0..ARRSIZEX, 0..ARRSIZEY, 0..ARRSIZEZ] OF BOOL;(* ~ 	(OPC : 1 : available for OPC-clients) *)
	{attribute 'OPC.UA.DA' := '1'}
	{attribute 'OPC.UA.DA.Description' := '3dim Array BOOL'}
	dyn_3dim_I1		: ARRAY[0..ARRSIZEX, 0..ARRSIZEY, 0..ARRSIZEZ] OF SINT;(* ~ 	(OPC : 1 : available for OPC-clients) *)
	{attribute 'OPC.UA.DA' := '1'}
	{attribute 'OPC.UA.DA.Description' := '3dim Array BOOL'}
	dyn_3dim_UI1	: ARRAY[0..ARRSIZEX, 0..ARRSIZEY, 0..ARRSIZEZ] OF USINT;(* ~ 	(OPC : 1 : available for OPC-clients) *)
	{attribute 'OPC.UA.DA' := '1'}
	{attribute 'OPC.UA.DA.Description' := '3dim Array BOOL'}
	dyn_3dim_I2 	: ARRAY[0..ARRSIZEX, 0..ARRSIZEY, 0..ARRSIZEZ] OF INT;(* ~ 	(OPC : 1 : available for OPC-clients) *)
	{attribute 'OPC.UA.DA' := '1'}
	{attribute 'OPC.UA.DA.Description' := '3dim Array BOOL'}
	dyn_3dim_UI2	: ARRAY[0..ARRSIZEX, 0..ARRSIZEY, 0..ARRSIZEZ] OF UINT;(* ~ 	(OPC : 1 : available for OPC-clients) *)
	{attribute 'OPC.UA.DA' := '1'}
	{attribute 'OPC.UA.DA.Description' := '3dim Array BOOL'}
	dyn_3dim_I4		: ARRAY[0..ARRSIZEX, 0..ARRSIZEY, 0..ARRSIZEZ] OF DINT;(* ~ 	(OPC : 1 : available for OPC-clients) *)
	{attribute 'OPC.UA.DA' := '1'}
	{attribute 'OPC.UA.DA.Description' := '3dim Array BOOL'}
	dyn_3dim_UI4	: ARRAY[0..ARRSIZEX, 0..ARRSIZEY, 0..ARRSIZEZ] OF UDINT;(* ~ 	(OPC : 1 : available for OPC-clients) *)
	{attribute 'OPC.UA.DA' := '1'}
	{attribute 'OPC.UA.DA.Description' := '3dim Array BOOL'}
	dyn_3dim_I8		: ARRAY[0..ARRSIZEX, 0..ARRSIZEY, 0..ARRSIZEZ] OF LINT;(* ~ 	(OPC : 1 : available for OPC-clients) *)
	{attribute 'OPC.UA.DA' := '1'}
	{attribute 'OPC.UA.DA.Description' := '3dim Array BOOL'}
	dyn_3dim_UI8	: ARRAY[0..ARRSIZEX, 0..ARRSIZEY, 0..ARRSIZEZ] OF ULINT;(* ~ 	(OPC : 1 : available for OPC-clients) *)
	{attribute 'OPC.UA.DA' := '1'}
	{attribute 'OPC.UA.DA.Description' := '3dim Array BOOL'}
	dyn_3dim_BYTE	: ARRAY[0..ARRSIZEX, 0..ARRSIZEY, 0..ARRSIZEZ] OF BYTE;(* ~ 	(OPC : 1 : available for OPC-clients) *)
	{attribute 'OPC.UA.DA' := '1'}
	{attribute 'OPC.UA.DA.Description' := '3dim Array BOOL'}
	dyn_3dim_WORD	: ARRAY[0..ARRSIZEX, 0..ARRSIZEY, 0..ARRSIZEZ] OF WORD;(* ~ 	(OPC : 1 : available for OPC-clients) *)
	{attribute 'OPC.UA.DA' := '1'}
	{attribute 'OPC.UA.DA.Description' := '3dim Array BOOL'}
	dyn_3dim_DWORD	: ARRAY[0..ARRSIZEX, 0..ARRSIZEY, 0..ARRSIZEZ] OF DWORD;(* ~ 	(OPC : 1 : available for OPC-clients) *)
	{attribute 'OPC.UA.DA' := '1'}
	{attribute 'OPC.UA.DA.Description' := '3dim Array BOOL'}
	dyn_3dim_LWORD	: ARRAY[0..ARRSIZEX, 0..ARRSIZEY, 0..ARRSIZEZ] OF LWORD;(* ~ 	(OPC : 1 : available for OPC-clients) *)
	{attribute 'OPC.UA.DA' := '1'}
	{attribute 'OPC.UA.DA.Description' := '3dim Array BOOL'}
	dyn_3dim_R4		: ARRAY[0..ARRSIZEX, 0..ARRSIZEY, 0..ARRSIZEZ] OF REAL;(* ~ 	(OPC : 1 : available for OPC-clients) *)
	{attribute 'OPC.UA.DA' := '1'}
	{attribute 'OPC.UA.DA.Description' := '3dim Array BOOL'}
	dyn_3dim_R8		: ARRAY[0..ARRSIZEX, 0..ARRSIZEY, 0..ARRSIZEZ] OF LREAL;(* ~ 	(OPC : 1 : available for OPC-clients) *)
	{attribute 'OPC.UA.DA' := '1'}
	{attribute 'OPC.UA.DA.Description' := '3dim Array BOOL'}
	dyn_3dim_BSTR	: ARRAY[0..ARRSIZEX, 0..ARRSIZEY, 0..ARRSIZEZ] OF STRING;(* ~ 	(OPC : 1 : available for OPC-clients) *)
	{attribute 'OPC.UA.DA' := '1'}
	{attribute 'OPC.UA.DA.Description' := '3dim Array BOOL'}
	//dyn_3dim_CHAR	: ARRAY[0..ARRSIZEX, 0..ARRSIZEY, 0..ARRSIZEZ] OF CHAR;(* ~ 	(OPC : 1 : available for OPC-clients) *)
	{attribute 'OPC.UA.DA' := '1'}
	{attribute 'OPC.UA.DA.Description' := '3dim Array BOOL'}
	dyn_3dim_WSTRING : ARRAY[0..ARRSIZEX, 0..ARRSIZEY, 0..ARRSIZEZ] OF WSTRING;(* ~ 	(OPC : 1 : available for OPC-clients) *)
	{attribute 'OPC.UA.DA' := '1'}
	{attribute 'OPC.UA.DA.Description' := '3dim Array BOOL'}
	//dyn_3dim_WCHAR: ARRAY[0..ARRSIZEX, 0..ARRSIZEY, 0..ARRSIZEZ] OF WCHAR;(* ~ 	(OPC : 1 : available for OPC-clients) *)
	{attribute 'OPC.UA.DA' := '1'}
	{attribute 'OPC.UA.DA.Description' := '3dim Array BOOL'}
	dyn_3dim_DT		: ARRAY[0..ARRSIZEX, 0..ARRSIZEY, 0..ARRSIZEZ] OF DT;(* ~ 	(OPC : 1 : available for OPC-clients) *)
	{attribute 'OPC.UA.DA' := '1'}
	{attribute 'OPC.UA.DA.Description' := '3dim Array BOOL'}
	dyn_3dim_DATE 	: ARRAY[0..ARRSIZEX, 0..ARRSIZEY, 0..ARRSIZEZ] OF DATE;(* ~ 	(OPC : 1 : available for OPC-clients) *)
	{attribute 'OPC.UA.DA' := '1'}
	{attribute 'OPC.UA.DA.Description' := '3dim Array BOOL'}
	dyn_3dim_TOD	: ARRAY[0..ARRSIZEX, 0..ARRSIZEY, 0..ARRSIZEZ] OF TOD;(* ~ 	(OPC : 1 : available for OPC-clients) *)
	{attribute 'OPC.UA.DA' := '1'}
	{attribute 'OPC.UA.DA.Description' := '3dim Array BOOL'}
	dyn_3dim_TIME	: ARRAY[0..ARRSIZEX, 0..ARRSIZEY, 0..ARRSIZEZ] OF TIME;(* ~ 	(OPC : 1 : available for OPC-clients) *)
END_VAR

// ---- GVLs/GVL_nodes_static.TcGVL
VAR_GLOBAL
	//scalars
	{attribute 'OPC.UA.DA' := '1'}
	{attribute 'OPC.UA.DA.Description' := 'Scalar LINT'}
	{attribute 'OPC.UA.DA.Access' := '1'}	
	stat_scalar_BOOL	: BOOL := TRUE;
	{attribute 'OPC.UA.DA' := '1'}
	{attribute 'OPC.UA.DA.Description' := 'Scalar SINT'}
	{attribute 'OPC.UA.DA.Access' := '1'}
	stat_scalar_I1		: SINT := 1;	
	{attribute 'OPC.UA.DA' := '1'}
	{attribute 'OPC.UA.DA.Description' := 'Scalar USINT'}
	{attribute 'OPC.UA.DA.Access' := '1'}
	stat_scalar_UI1		: USINT := 1;	
	{attribute 'OPC.UA.DA' := '1'}
	{attribute 'OPC.UA.DA.Description' := 'Scalar INT'}
	{attribute 'OPC.UA.DA.Access' := '1'}
	stat_scalar_I2 		: INT := 1;		
	{attribute 'OPC.UA.DA' := '1'}
	{attribute 'OPC.UA.DA.Description' := 'Scalar UINT'}
	{attribute 'OPC.UA.DA.Access' := '1'}
	stat_scalar_UI2		: UINT := 1;	
	{attribute 'OPC.UA.DA' := '1'}
	{attribute 'OPC.UA.DA.Description' := 'Scalar DINT'}
	{attribute 'OPC.UA.DA.Access' := '1'}
	stat_scalar_I4		: DINT := 1;	
	{attribute 'OPC.UA.DA' := '1'}
	{attribute 'OPC.UA.DA.Description' := 'Scalar UDINT'}
	{attribute 'OPC.UA.DA.Access' := '1'}
	stat_scalar_UI4		: UDINT := 1;	
	{attribute 'OPC.UA.DA' := '1'}
	{attribute 'OPC.UA.DA.Description' := 'Scalar LINT'}
	{attribute 'OPC.UA.DA.Access' := '1'}
	stat_scalar_I8		: LINT := 1;	
	{attribute 'OPC.UA.DA' := '1'}
	{attribute 'OPC.UA.DA.Description' := 'Scalar ULINT'}
	{attribute 'OPC.UA.DA.Access' := '1'}
	stat_scalar_UI8		: ULINT := 1;	
	{attribute 'OPC.UA.DA' := '1'}
	{attribute 'OPC.UA.DA.Description' := 'Scalar BYTE'}
	{attribute 'OPC.UA.DA.Access' := '1'}
	stat_scalar_BYTE	: BYTE := 1;	
	{attribute 'OPC.UA.DA' := '1'}
	{attribute 'OPC.UA.DA.Description' := 'Scalar WORD'}
	{attribute 'OPC.UA.DA.Access' := '1'}
	stat_scalar_WORD	: WORD := 1;	
	{attribute 'OPC.UA.DA' := '1'}
	{attribute 'OPC.UA.DA.Description' := 'Scalar DWORD'}
	{attribute 'OPC.UA.DA.Access' := '1'}
	stat_scalar_DWORD	: DWORD := 1;	
	{attribute 'OPC.UA.DA' := '1'}
	{attribute 'OPC.UA.DA.Description' := 'Scalar LWORD'}
	{attribute 'OPC.UA.DA.Access' := '1'}
	stat_scalar_LWORD	: LWORD := 1;				
	{attribute 'OPC.UA.DA' := '1'}
	{attribute 'OPC.UA.DA.Description' := 'Scalar REAL'}
	{attribute 'OPC.UA.DA.Access' := '1'}
	stat_scalar_R4		: REAL := 1.0;				
	{attribute 'OPC.UA.DA' := '1'}
	{attribute 'OPC.UA.DA.Description' := 'Scalar LREAL'}
	{attribute 'OPC.UA.DA.Access' := '1'}
	stat_scalar_R8		: LREAL := 1.0;				
	{attribute 'OPC.UA.DA' := '1'}
	{attribute 'OPC.UA.DA.Description' := 'Scalar STRING'}
	{attribute 'OPC.UA.DA.Access' := '1'}
	stat_scalar_BSTR	: STRING := 'Hello World';
	{attribute 'OPC.UA.DA' := '1'}
	{attribute 'OPC.UA.DA.Description' := 'Scalar WSTRING'}
	{attribute 'OPC.UA.DA.Access' := '1'}
	stat_scalar_WSTRING	: WSTRING := "Hello World";
	{attribute 'OPC.UA.DA' := '1'}
	{attribute 'OPC.UA.DA.Description' := 'Scalar DT'}
	{attribute 'OPC.UA.DA.Access' := '1'}
	stat_scalar_DT		: DT;
	{attribute 'OPC.UA.DA' := '1'}
	{attribute 'OPC.UA.DA.Description' := 'Scalar DATE'}
	{attribute 'OPC.UA.DA.Access' := '1'}
	stat_scalar_DATE 	: DATE;
	{attribute 'OPC.UA.DA' := '1'}
	{attribute 'OPC.UA.DA.Description' := 'Scalar TOD'}
	{attribute 'OPC.UA.DA.Access' := '1'}
	stat_scalar_TOD		: TOD;	
	{attribute 'OPC.UA.DA' := '1'}
	{attribute 'OPC.UA.DA.Description' := 'Scalar TIME'}
	{attribute 'OPC.UA.DA.Access' := '1'}
	stat_scalar_TIME	: TIME;	

	
	//1dim
	{attribute 'OPC.UA.DA' := '1'}
	{attribute 'OPC.UA.DA.Description' := '1dim Array BOOL'}
	{attribute 'OPC.UA.DA.Access' := '1'}	
	stat_1dim_BOOL		: ARRAY[0..ARRSIZEX] OF BOOL;
	{attribute 'OPC.UA.DA' := '1'}
	{attribute 'OPC.UA.DA.Description' := '1dim Array SINT'}
	{attribute 'OPC.UA.DA.Access' := '1'}
	stat_1dim_I1		: ARRAY[0..ARRSIZEX] OF SINT;
	{attribute 'OPC.UA.DA' := '1'}
	{attribute 'OPC.UA.DA.Description' := '1dim Array USINT'}
	{attribute 'OPC.UA.DA.Access' := '1'}
	stat_1dim_UI1		: ARRAY[0..ARRSIZEX] OF USINT;
	{attribute 'OPC.UA.DA' := '1'}
	{attribute 'OPC.UA.DA.Description' := '1dim Array INT'}
	{attribute 'OPC.UA.DA.Access' := '1'}
	stat_1dim_I2 		: ARRAY[0..ARRSIZEX] OF INT;	
	{attribute 'OPC.UA.DA' := '1'}
	{attribute 'OPC.UA.DA.Description' := '1dim Array UINT'}
	{attribute 'OPC.UA.DA.Access' := '1'}
	stat_1dim_UI2		: ARRAY[0..ARRSIZEX] OF UINT;
	{attribute 'OPC.UA.DA' := '1'}
	{attribute 'OPC.UA.DA.Description' := '1dim Array DINT'}
	{attribute 'OPC.UA.DA.Access' := '1'}
	stat_1dim_I4		: ARRAY[0..ARRSIZEX] OF DINT;
	{attribute 'OPC.UA.DA' := '1'}
	{attribute 'OPC.UA.DA.Description' := '1dim Array UDINT'}
	{attribute 'OPC.UA.DA.Access' := '1'}
	stat_1dim_UI4		: ARRAY[0..ARRSIZEX] OF UDINT;
	{attribute 'OPC.UA.DA' := '1'}
	{attribute 'OPC.UA.DA.Description' := '1dim Array LINT'}
	{attribute 'OPC.UA.DA.Access' := '1'}
	stat_1dim_I8		: ARRAY[0..ARRSIZEX] OF LINT;
	{attribute 'OPC.UA.DA' := '1'}
	{attribute 'OPC.UA.DA.Description' := '1dim Array ULINT'}
	{attribute 'OPC.UA.DA.Access' := '1'}
	stat_1dim_UI8		: ARRAY[0..ARRSIZEX] OF ULINT;
	{attribute 'OPC.UA.DA' := '1'}
	{attribute 'OPC.UA.DA.Description' := '1dim Array BYTE'}
	{attribute 'OPC.UA.DA.Access' := '1'}
	stat_1dim_BYTE		: ARRAY[0..ARRSIZEX] OF BYTE;
	{attribute 'OPC.UA.DA' := '1'}
	{attribute 'OPC.UA.DA.Description' := '1dim Array WORD'}
	{attribute 'OPC.UA.DA.Access' := '1'}
	stat_1dim_WORD		: ARRAY[0..ARRSIZEX] OF WORD;
	{attribute 'OPC.UA.DA' := '1'}
	{attribute 'OPC.UA.DA.Description' := '1dim Array DWORD'}
	{attribute 'OPC.UA.DA.Access' := '1'}
	stat_1dim_DWORD		: ARRAY[0..ARRSIZEX] OF DWORD;
	{attribute 'OPC.UA.DA' := '1'}
	{attribute 'OPC.UA.DA.Description' := '1dim Array LWORD'}
	{attribute 'OPC.UA.DA.Access' := '1'}
	stat_1dim_LWORD		: ARRAY[0..ARRSIZEX] OF LWORD;
	{attribute 'OPC.UA.DA' := '1'}
	{attribute 'OPC.UA.DA.Description' := '1dim Array REAL'}
	{attribute 'OPC.UA.DA.Access' := '1'}
	stat_1dim_R4		: ARRAY[0..ARRSIZEX] OF REAL;
	{attribute 'OPC.UA.DA' := '1'}
	{attribute 'OPC.UA.DA.Description' := '1dim Array LREAL'}
	{attribute 'OPC.UA.DA.Access' := '1'}
	stat_1dim_R8		: ARRAY[0..ARRSIZEX] OF LREAL;
	{attribute 'OPC.UA.DA' := '1'}
	{attribute 'OPC.UA.DA.Description' := '1dim Array STRING'}
	{attribute 'OPC.UA.DA.Access' := '1'}
	stat_1dim_BSTR		: ARRAY[0..ARRSIZEX] OF STRING;
	{attribute 'OPC.UA.DA' := '1'}
	{attribute 'OPC.UA.DA.Description' := '1dim Array WSTRING'}
	{attribute 'OPC.UA.DA.Access' := '1'}
	stat_1dim_WSTRING	: ARRAY[0..ARRSIZEX] OF WSTRING;
	{attribute 'OPC.UA.DA' := '1'}
	{attribute 'OPC.UA.DA.Description' := '1dim Array DT'}
	{attribute 'OPC.UA.DA.Access' := '1'}
	stat_1dim_DT		: ARRAY[0..ARRSIZEX] OF DT;		
	{attribute 'OPC.UA.DA' := '1'}
	{attribute 'OPC.UA.DA.Description' := '1dim Array DATE'}
	{attribute 'OPC.UA.DA.Access' := '1'}
	stat_1dim_DATE 		: ARRAY[0..ARRSIZEX] OF DATE;	
	{attribute 'OPC.UA.DA' := '1'}
	{attribute 'OPC.UA.DA.Description' := '1dim Array TOD'}
	{attribute 'OPC.UA.DA.Access' := '1'}
	stat_1dim_TOD		: ARRAY[0..ARRSIZEX] OF TOD;	
	{attribute 'OPC.UA.DA' := '1'}
	{attribute 'OPC.UA.DA.Description' := '1dim Array TIME'}
	{attribute 'OPC.UA.DA.Access' := '1'}
	stat_1dim_TIME		: ARRAY[0..ARRSIZEX] OF TIME;	

	
	//2dim
	{attribute 'OPC.UA.DA' := '1'}
	{attribute 'OPC.UA.DA.Description' := '2dim Array BOOL'}
	stat_2dim_BOOL		: ARRAY[0..ARRSIZEX, 0..ARRSIZEY] OF BOOL;
	{attribute 'OPC.UA.DA' := '1'}
	{attribute 'OPC.UA.DA.Description' := '2dim Array SINT'}
	stat_2dim_I1		: ARRAY[0..ARRSIZEX, 0..ARRSIZEY] OF SINT;
	{attribute 'OPC.UA.DA' := '1'}
	{attribute 'OPC.UA.DA.Description' := '2dim Array USINT'}
	stat_2dim_UI1		: ARRAY[0..ARRSIZEX, 0..ARRSIZEY] OF USINT;
	{attribute 'OPC.UA.DA' := '1'}
	{attribute 'OPC.UA.DA.Description' := '2dim Array INT'}
	stat_2dim_I2 		: ARRAY[0..ARRSIZEX, 0..ARRSIZEY] OF INT;
	{attribute 'OPC.UA.DA' := '1'}
	{attribute 'OPC.UA.DA.Description' := '2dim Array UINT'}
	stat_2dim_UI2		: ARRAY[0..ARRSIZEX, 0..ARRSIZEY] OF UINT;
	{attribute 'OPC.UA.DA' := '1'}
	{attribute 'OPC.UA.DA.Description' := '2dim Array DINT'}
	stat_2dim_I4		: ARRAY[0..ARRSIZEX, 0..ARRSIZEY] OF DINT;
	{attribute 'OPC.UA.DA' := '1'}
	{attribute 'OPC.UA.DA.Description' := '2dim Array UDINT'}
	stat_2dim_UI4		: ARRAY[0..ARRSIZEX, 0..ARRSIZEY] OF UDINT;
	{attribute 'OPC.UA.DA' := '1'}
	{attribute 'OPC.UA.DA.Description' := '2dim Array LINT'}
	stat_2dim_I8		: ARRAY[0..ARRSIZEX, 0..ARRSIZEY] OF LINT;	
	{attribute 'OPC.UA.DA' := '1'}
	{attribute 'OPC.UA.DA.Description' := '2dim Array ULINT'}
	stat_2dim_UI8		: ARRAY[0..ARRSIZEX, 0..ARRSIZEY] OF ULINT;
	{attribute 'OPC.UA.DA' := '1'}
	{attribute 'OPC.UA.DA.Description' := '2dim Array BYTE'}
	stat_2dim_BYTE		: ARRAY[0..ARRSIZEX, 0..ARRSIZEY] OF BYTE;	
	{attribute 'OPC.UA.DA' := '1'}
	{attribute 'OPC.UA.DA.Description' := '2dim Array WORD'}
	stat_2dim_WORD		: ARRAY[0..ARRSIZEX, 0..ARRSIZEY] OF WORD;	
	{attribute 'OPC.UA.DA' := '1'}
	{attribute 'OPC.UA.DA.Description' := '2dim Array DWORD'}
	stat_2dim_DWORD		: ARRAY[0..ARRSIZEX, 0..ARRSIZEY] OF DWORD;	
	{attribute 'OPC.UA.DA' := '1'}
	{attribute 'OPC.UA.DA.Description' := '2dim Array LWORD'}
	stat_2dim_LWORD		: ARRAY[0..ARRSIZEX, 0..ARRSIZEY] OF LWORD;
	{attribute 'OPC.UA.DA' := '1'}
	{attribute 'OPC.UA.DA.Description' := '2dim Array REAL'}
	stat_2dim_R4		: ARRAY[0..ARRSIZEX, 0..ARRSIZEY] OF REAL;
	{attribute 'OPC.UA.DA' := '1'}
	{attribute 'OPC.UA.DA.Description' := '2dim Array LREAL'}
	stat_2dim_R8		: ARRAY[0..ARRSIZEX, 0..ARRSIZEY] OF LREAL;
	{attribute 'OPC.UA.DA' := '1'}
	{attribute 'OPC.UA.DA.Description' := '2dim Array STRING'}
	stat_2dim_BSTR		: ARRAY[0..ARRSIZEX, 0..ARRSIZEY] OF STRING;
	{attribute 'OPC.UA.DA' := '1'}
	{attribute 'OPC.UA.DA.Description' := '2dim Array WSTRING'}
	stat_2dim_WSTRING	: ARRAY[0..ARRSIZEX, 0..ARRSIZEY] OF WSTRING;
	{attribute 'OPC.UA.DA' := '1'}
	{attribute 'OPC.UA.DA.Description' := '2dim Array DT'}
	stat_2dim_DT		: ARRAY[0..ARRSIZEX, 0..ARRSIZEY] OF DT;
	{attribute 'OPC.UA.DA' := '1'}
	{attribute 'OPC.UA.DA.Description' := '2dim Array DATE'}
	stat_2dim_DATE	 	: ARRAY[0..ARRSIZEX, 0..ARRSIZEY] OF DATE;
	{attribute 'OPC.UA.DA' := '1'}
	{attribute 'OPC.UA.DA.Description' := '2dim Array TOD'}
	stat_2dim_TOD		: ARRAY[0..ARRSIZEX, 0..ARRSIZEY] OF TOD;
	{attribute 'OPC.UA.DA' := '1'}
	{attribute 'OPC.UA.DA.Description' := '2dim Array TIME'}
	stat_2dim_TIME		: ARRAY[0..ARRSIZEX, 0..ARRSIZEY] OF TIME;

	//3dim
	{attribute 'OPC.UA.DA' := '1'}
	{attribute 'OPC.UA.DA.Description' := '3dim Array BOOL'}
	stat_3dim_BOOL		: ARRAY[0..ARRSIZEX, 0..ARRSIZEY, 0..ARRSIZEZ] OF BOOL;
	{attribute 'OPC.UA.DA' := '1'}
	{attribute 'OPC.UA.DA.Description' := '3dim Array SINT'}
	stat_3dim_I1		: ARRAY[0..ARRSIZEX, 0..ARRSIZEY, 0..ARRSIZEZ] OF SINT;
	{attribute 'OPC.UA.DA' := '1'}
	{attribute 'OPC.UA.DA.Description' := '3dim Array USINT'}
	stat_3dim_UI1		: ARRAY[0..ARRSIZEX, 0..ARRSIZEY, 0..ARRSIZEZ] OF USINT;
	{attribute 'OPC.UA.DA' := '1'}
	{attribute 'OPC.UA.DA.Description' := '3dim Array INT'}
	stat_3dim_I2 		: ARRAY[0..ARRSIZEX, 0..ARRSIZEY, 0..ARRSIZEZ] OF INT;
	{attribute 'OPC.UA.DA' := '1'}
	{attribute 'OPC.UA.DA.Description' := '3dim Array UINT'}
	stat_3dim_UI2		: ARRAY[0..ARRSIZEX, 0..ARRSIZEY, 0..ARRSIZEZ] OF UINT;
	{attribute 'OPC.UA.DA' := '1'}
	{attribute 'OPC.UA.DA.Description' := '3dim Array DINT'}
	stat_3dim_I4		: ARRAY[0..ARRSIZEX, 0..ARRSIZEY, 0..ARRSIZEZ] OF DINT;
	{attribute 'OPC.UA.DA' := '1'}
	{attribute 'OPC.UA.DA.Description' := '3dim Array UDINT'}
	stat_3dim_UI4		: ARRAY[0..ARRSIZEX, 0..ARRSIZEY, 0..ARRSIZEZ] OF UDINT;
	{attribute 'OPC.UA.DA' := '1'}
	{attribute 'OPC.UA.DA.Description' := '3dim Array LINT'}
	stat_3dim_I8		: ARRAY[0..ARRSIZEX, 0..ARRSIZEY, 0..ARRSIZEZ] OF LINT;
	{attribute 'OPC.UA.DA' := '1'}
	{attribute 'OPC.UA.DA.Description' := '3dim Array ULINT'}
	stat_3dim_UI8		: ARRAY[0..ARRSIZEX, 0..ARRSIZEY, 0..ARRSIZEZ] OF ULINT;
	{attribute 'OPC.UA.DA' := '1'}
	{attribute 'OPC.UA.DA.Description' := '3dim Array BYTE'}
	stat_3dim_BYTE		: ARRAY[0..ARRSIZEX, 0..ARRSIZEY, 0..ARRSIZEZ] OF BYTE;
	{attribute 'OPC.UA.DA' := '1'}
	{attribute 'OPC.UA.DA.Description' := '3dim Array WORD'}
	stat_3dim_WORD		: ARRAY[0..ARRSIZEX, 0..ARRSIZEY, 0..ARRSIZEZ] OF WORD;
	{attribute 'OPC.UA.DA' := '1'}
	{attribute 'OPC.UA.DA.Description' := '3dim Array DWORD'}
	stat_3dim_DWORD		: ARRAY[0..ARRSIZEX, 0..ARRSIZEY, 0..ARRSIZEZ] OF DWORD;
	{attribute 'OPC.UA.DA' := '1'}
	{attribute 'OPC.UA.DA.Description' := '3dim Array LWORD'}
	stat_3dim_LWORD		: ARRAY[0..ARRSIZEX, 0..ARRSIZEY, 0..ARRSIZEZ] OF LWORD;
	{attribute 'OPC.UA.DA' := '1'}
	{attribute 'OPC.UA.DA.Description' := '3dim Array REAL'}
	stat_3dim_R4		: ARRAY[0..ARRSIZEX, 0..ARRSIZEY, 0..ARRSIZEZ] OF REAL;	
	{attribute 'OPC.UA.DA' := '1'}
	{attribute 'OPC.UA.DA.Description' := '3dim Array LREAL'}
	stat_3dim_R8		: ARRAY[0..ARRSIZEX, 0..ARRSIZEY, 0..ARRSIZEZ] OF LREAL;
	{attribute 'OPC.UA.DA' := '1'}
	{attribute 'OPC.UA.DA.Description' := '3dim Array STRING'}
	stat_3dim_BSTR		: ARRAY[0..ARRSIZEX, 0..ARRSIZEY, 0..ARRSIZEZ] OF STRING;
	{attribute 'OPC.UA.DA' := '1'}
	{attribute 'OPC.UA.DA.Description' := '3dim Array WSTRING'}
	stat_3dim_WSTRING 	: ARRAY[0..ARRSIZEX, 0..ARRSIZEY, 0..ARRSIZEZ] OF WSTRING;
	{attribute 'OPC.UA.DA' := '1'}
	{attribute 'OPC.UA.DA.Description' := '3dim Array DT'}
	stat_3dim_DT		: ARRAY[0..ARRSIZEX, 0..ARRSIZEY, 0..ARRSIZEZ] OF DT;
	{attribute 'OPC.UA.DA' := '1'}
	{attribute 'OPC.UA.DA.Description' := '3dim Array DATE'}
	stat_3dim_DATE 		: ARRAY[0..ARRSIZEX, 0..ARRSIZEY, 0..ARRSIZEZ] OF DATE;
	{attribute 'OPC.UA.DA' := '1'}
	{attribute 'OPC.UA.DA.Description' := '3dim Array TOD'}
	stat_3dim_TOD		: ARRAY[0..ARRSIZEX, 0..ARRSIZEY, 0..ARRSIZEZ] OF TOD;	
	{attribute 'OPC.UA.DA' := '1'}
	{attribute 'OPC.UA.DA.Description' := '3dim Array TIME'}
	stat_3dim_TIME		: ARRAY[0..ARRSIZEX, 0..ARRSIZEY, 0..ARRSIZEZ] OF TIME;

	
	// Scalars writeable
	{attribute 'OPC.UA.DA' := '1'}
	{attribute 'OPC.UA.DA.Description' := 'Scalar LINT'}	
	stat_scalar_BOOL_writeable	: BOOL := TRUE;
	{attribute 'OPC.UA.DA' := '1'}
	{attribute 'OPC.UA.DA.Description' := 'Scalar SINT'}
	stat_scalar_I1_writeable		: SINT := 1;	
	{attribute 'OPC.UA.DA' := '1'}
	{attribute 'OPC.UA.DA.Description' := 'Scalar USINT'}
	stat_scalar_UI1_writeable		: USINT := 1;	
	{attribute 'OPC.UA.DA' := '1'}
	{attribute 'OPC.UA.DA.Description' := 'Scalar INT'}
	stat_scalar_I2_writeable 		: INT := 1;		
	{attribute 'OPC.UA.DA' := '1'}
	{attribute 'OPC.UA.DA.Description' := 'Scalar UINT'}
	stat_scalar_UI2_writeable		: UINT := 1;	
	{attribute 'OPC.UA.DA' := '1'}
	{attribute 'OPC.UA.DA.Description' := 'Scalar DINT'}
	stat_scalar_I4_writeable		: DINT := 1;	
	{attribute 'OPC.UA.DA' := '1'}
	{attribute 'OPC.UA.DA.Description' := 'Scalar UDINT'}
	stat_scalar_UI4_writeable		: UDINT := 1;	
	{attribute 'OPC.UA.DA' := '1'}
	{attribute 'OPC.UA.DA.Description' := 'Scalar LINT'}
	stat_scalar_I8_writeable		: LINT := 1;	
	{attribute 'OPC.UA.DA' := '1'}
	{attribute 'OPC.UA.DA.Description' := 'Scalar ULINT'}
	stat_scalar_UI8_writeable		: ULINT := 1;	
	{attribute 'OPC.UA.DA' := '1'}
	{attribute 'OPC.UA.DA.Description' := 'Scalar BYTE'}
	stat_scalar_BYTE_writeable	: BYTE := 1;	
	{attribute 'OPC.UA.DA' := '1'}
	{attribute 'OPC.UA.DA.Description' := 'Scalar WORD'}
	stat_scalar_WORD_writeable	: WORD := 1;	
	{attribute 'OPC.UA.DA' := '1'}
	{attribute 'OPC.UA.DA.Description' := 'Scalar DWORD'}
	stat_scalar_DWORD_writeable	: DWORD := 1;	
	{attribute 'OPC.UA.DA' := '1'}
	{attribute 'OPC.UA.DA.Description' := 'Scalar LWORD'}
	stat_scalar_LWORD_writeable	: LWORD := 1;				
	{attribute 'OPC.UA.DA' := '1'}
	{attribute 'OPC.UA.DA.Description' := 'Scalar REAL'}
	stat_scalar_R4_writeable		: REAL := 1.0;				
	{attribute 'OPC.UA.DA' := '1'}
	{attribute 'OPC.UA.DA.Description' := 'Scalar LREAL'}
	stat_scalar_R8_writeable		: LREAL := 1.0;				
	{attribute 'OPC.UA.DA' := '1'}
	{attribute 'OPC.UA.DA.Description' := 'Scalar STRING'}
	stat_scalar_BSTR_writeable	: STRING := 'Hello World';
	{attribute 'OPC.UA.DA' := '1'}
	{attribute 'OPC.UA.DA.Description' := 'Scalar WSTRING'}
	stat_scalar_WSTRING_writeable	: WSTRING := "Hello World";
	{attribute 'OPC.UA.DA' := '1'}
	{attribute 'OPC.UA.DA.Description' := 'Scalar DT'}
	stat_scalar_DT_writeable		: DT;
	{attribute 'OPC.UA.DA' := '1'}
	{attribute 'OPC.UA.DA.Description' := 'Scalar DATE'}
	stat_scalar_DATE_writeable 	: DATE;
	{attribute 'OPC.UA.DA' := '1'}
	{attribute 'OPC.UA.DA.Description' := 'Scalar TOD'}
	stat_scalar_TOD_writeable		: TOD;	
	{attribute 'OPC.UA.DA' := '1'}
	{attribute 'OPC.UA.DA.Description' := 'Scalar TIME'}
	stat_scalar_TIME_writeable	: TIME;	

	
	//1dim
	{attribute 'OPC.UA.DA' := '1'}
	{attribute 'OPC.UA.DA.Description' := '1dim Array BOOL'}	
	stat_1dim_BOOL_writeable		: ARRAY[0..ARRSIZEX] OF BOOL;
	{attribute 'OPC.UA.DA' := '1'}
	{attribute 'OPC.UA.DA.Description' := '1dim Array SINT'}
	stat_1dim_I1_writeable		: ARRAY[0..ARRSIZEX] OF SINT;
	{attribute 'OPC.UA.DA' := '1'}
	{attribute 'OPC.UA.DA.Description' := '1dim Array USINT'}
	stat_1dim_UI1_writeable		: ARRAY[0..ARRSIZEX] OF USINT;
	{attribute 'OPC.UA.DA' := '1'}
	{attribute 'OPC.UA.DA.Description' := '1dim Array INT'}
	stat_1dim_I2_writeable 		: ARRAY[0..ARRSIZEX] OF INT;	
	{attribute 'OPC.UA.DA' := '1'}
	{attribute 'OPC.UA.DA.Description' := '1dim Array UINT'}
	stat_1dim_UI2_writeable		: ARRAY[0..ARRSIZEX] OF UINT;
	{attribute 'OPC.UA.DA' := '1'}
	{attribute 'OPC.UA.DA.Description' := '1dim Array DINT'}
	stat_1dim_I4_writeable		: ARRAY[0..ARRSIZEX] OF DINT;
	{attribute 'OPC.UA.DA' := '1'}
	{attribute 'OPC.UA.DA.Description' := '1dim Array UDINT'}
	stat_1dim_UI4_writeable		: ARRAY[0..ARRSIZEX] OF UDINT;
	{attribute 'OPC.UA.DA' := '1'}
	{attribute 'OPC.UA.DA.Description' := '1dim Array LINT'}
	stat_1dim_I8_writeable		: ARRAY[0..ARRSIZEX] OF LINT;
	{attribute 'OPC.UA.DA' := '1'}
	{attribute 'OPC.UA.DA.Description' := '1dim Array ULINT'}
	stat_1dim_UI8_writeable		: ARRAY[0..ARRSIZEX] OF ULINT;
	{attribute 'OPC.UA.DA' := '1'}
	{attribute 'OPC.UA.DA.Description' := '1dim Array BYTE'}
	stat_1dim_BYTE_writeable		: ARRAY[0..ARRSIZEX] OF BYTE;
	{attribute 'OPC.UA.DA' := '1'}
	{attribute 'OPC.UA.DA.Description' := '1dim Array WORD'}
	stat_1dim_WORD_writeable		: ARRAY[0..ARRSIZEX] OF WORD;
	{attribute 'OPC.UA.DA' := '1'}
	{attribute 'OPC.UA.DA.Description' := '1dim Array DWORD'}
	stat_1dim_DWORD_writeable		: ARRAY[0..ARRSIZEX] OF DWORD;
	{attribute 'OPC.UA.DA' := '1'}
	{attribute 'OPC.UA.DA.Description' := '1dim Array LWORD'}
	stat_1dim_LWORD_writeable		: ARRAY[0..ARRSIZEX] OF LWORD;
	{attribute 'OPC.UA.DA' := '1'}
	{attribute 'OPC.UA.DA.Description' := '1dim Array REAL'}
	stat_1dim_R4_writeable		: ARRAY[0..ARRSIZEX] OF REAL;
	{attribute 'OPC.UA.DA' := '1'}
	{attribute 'OPC.UA.DA.Description' := '1dim Array LREAL'}
	stat_1dim_R8_writeable		: ARRAY[0..ARRSIZEX] OF LREAL;
	{attribute 'OPC.UA.DA' := '1'}
	{attribute 'OPC.UA.DA.Description' := '1dim Array STRING'}
	stat_1dim_BSTR_writeable		: ARRAY[0..ARRSIZEX] OF STRING;
	{attribute 'OPC.UA.DA' := '1'}
	{attribute 'OPC.UA.DA.Description' := '1dim Array WSTRING'}
	stat_1dim_WSTRING_writeable	: ARRAY[0..ARRSIZEX] OF WSTRING;
	{attribute 'OPC.UA.DA' := '1'}
	{attribute 'OPC.UA.DA.Description' := '1dim Array DT'}
	stat_1dim_DT_writeable		: ARRAY[0..ARRSIZEX] OF DT;		
	{attribute 'OPC.UA.DA' := '1'}
	{attribute 'OPC.UA.DA.Description' := '1dim Array DATE'}
	stat_1dim_DATE_writeable 		: ARRAY[0..ARRSIZEX] OF DATE;	
	{attribute 'OPC.UA.DA' := '1'}
	{attribute 'OPC.UA.DA.Description' := '1dim Array TOD'}
	stat_1dim_TOD_writeable		: ARRAY[0..ARRSIZEX] OF TOD;	
	{attribute 'OPC.UA.DA' := '1'}
	{attribute 'OPC.UA.DA.Description' := '1dim Array TIME'}
	stat_1dim_TIME_writeable		: ARRAY[0..ARRSIZEX] OF TIME;		
END_VAR

// ---- POUs/MAIN.TcPOU
PROGRAM MAIN
VAR
	bInit : BOOL := TRUE;	
END_VAR

(* Static values and namespace test are initialized only once upon startup *)
IF bInit THEN
	bInit := FALSE;
	PRG_Static();
END_IF
PRG_Dynamic(); // Data generation for variables in GVL_nodes_dynamic
PRG_Eventlogger(); // Sample for TcEventlogger integration
PRG_HistoricalAccess(); // Data generation for variables in GVL_historizing (Historical Access)
PRG_AlarmsConditions(); // Data generation for variables in GVL_alarms_condition (Alarms & Conditions)
PRG_Methods(); // Includes methods

END_PROGRAM

// ---- POUs/Programs/PRG_Static.TcPOU
(* This program initializes variable values from GVL_nodes_static and GVL_structures to a static value that does not change during runtime. *)
PROGRAM PRG_Static
VAR
	k: INT;
	l: INT;
	m: INT;
END_VAR

	stat_scalar_BOOL	:= TRUE;
	stat_scalar_I1		:= 1;	
	stat_scalar_UI1		:= 1;	
	stat_scalar_I2 		:= 1;		
	stat_scalar_UI2		:= 1;	
	stat_scalar_I4		:= 1;	
	stat_scalar_UI4		:= 1;	
	stat_scalar_I8		:= 1;	
	stat_scalar_UI8		:= 1;	
	stat_scalar_BYTE	:= 1;	
	stat_scalar_WORD	:= 1;	
	stat_scalar_DWORD	:= 1;	
	stat_scalar_LWORD	:= 1;				
	stat_scalar_R4		:= 1.0;				
	stat_scalar_R8		:= 1.0;				
	stat_scalar_BSTR	:= 'Hello World';
	stat_scalar_WSTRING	:= "Hello World";
	stat_scalar_DT		:= DT#1972-03-29-00:00:00;
	stat_scalar_DATE 	:= DATE#1972-03-29;
	stat_scalar_TOD		:= TOD#12:00:00;	
	stat_scalar_TIME	:= T#1S;	

	GVL_structures.StructuredType1.a 			:= 42;
	GVL_structures.StructuredType1.b			:= 42;
	GVL_structures.StructuredType1.x			:= E_Enum_1.THREE;
	GVL_structures.StructuredType1.str			:= 'Hello World';

	GVL_structures.StructuredType2.c1.a			:= 42;
	GVL_structures.StructuredType2.c1.b			:= 42;
	GVL_structures.StructuredType2.c1.x			:= E_Enum_1.THREE;
	GVL_structures.StructuredType2.c1.str		:= 'Hello World';
	GVL_structures.StructuredType2.s_5			:= 'Hello';
	GVL_structures.StructuredType2.s_3			:= 'Hel';
	FOR k:= 0 TO 5 DO
		GVL_structures.StructuredType2.cArr[k].a:= 42;
		GVL_structures.StructuredType2.cArr[k].b:= 42;
		GVL_structures.StructuredType2.cArr[k].x:= E_Enum_1.THREE;
		GVL_structures.StructuredType2.cArr[k].str:= 'Hello World'; 
	END_FOR	
	GVL_structures.StructuredType2.e			:= E_Enum_1.THREE;
	FOR k:= 0 TO 100 DO
		GVL_structures.StructuredType2.iArr[k] := 42;
	END_FOR
	
	GVL_structures.StructuredType8.stComplex.a			:= 42;
	GVL_structures.StructuredType8.stComplex.b			:= 42;
	GVL_structures.StructuredType8.stComplex.x			:= E_Enum_1.THREE;
	GVL_structures.StructuredType8.stComplex.str		:= 'Hello World';
	GVL_structures.StructuredType8.strString5			:= 'Hello';
	GVL_structures.StructuredType8.strString3			:= 'Hel';
	FOR k:= 0 TO 1 DO
		GVL_structures.StructuredType8.arrComplex[k].a:= 42;
		GVL_structures.StructuredType8.arrComplex[k].b:= 42;
		GVL_structures.StructuredType8.arrComplex[k].x:= E_Enum_1.THREE;
		GVL_structures.StructuredType8.arrComplex[k].str:= 'Hello World'; 
	END_FOR	
	GVL_structures.StructuredType8.eEnum			:= E_Enum_1.THREE;
	FOR k:= 0 TO 100 DO
		GVL_structures.StructuredType8.arrDint[k] := 42;
	END_FOR	
	
	FOR k:= 0 TO ARRSIZEX DO
		stat_1dim_BOOL[k] := TRUE;
		stat_1dim_I1[k] := 1;
		stat_1dim_UI1[k] := 1;
		stat_1dim_I2[k] := 1;
		stat_1dim_UI2[k] := 1;
		stat_1dim_I4[k] := 1;
		stat_1dim_UI4[k] := 1;
		stat_1dim_I8[k] := 1;
		stat_1dim_UI8[k] := 1;
		stat_1dim_BYTE[k] := 1;
		stat_1dim_WORD[k] := 1;
		stat_1dim_DWORD[k] := 1;
		stat_1dim_LWORD[k] := 1;
		stat_1dim_R4[k] := 1.0;
		stat_1dim_R8[k] := 1.0;
		stat_1dim_BSTR[k] := 'Hello World';
		stat_1dim_WSTRING[k] := "Hello World";
		stat_1dim_DT[k] := DT#1972-03-29-00:00:00;
		stat_1dim_DATE[k] := DATE#1972-03-29;
		stat_1dim_TOD[k] := TOD#12:00:00;
		stat_1dim_TIME[k] := T#1S;
	END_FOR	

FOR l:= 0 TO ARRSIZEY DO
	FOR k:= 0 TO ARRSIZEX DO
		stat_2dim_BOOL[k,l] := TRUE;
		stat_2dim_I1[k,l] := 1;
		stat_2dim_UI1[k,l] := 1;
		stat_2dim_I2[k,l] := 1;
		stat_2dim_UI2[k,l] := 1;
		stat_2dim_I4[k,l] := 1;
		stat_2dim_UI4[k,l] := 1;
		stat_2dim_I8[k,l] := 1;
		stat_2dim_UI8[k,l] := 1;
		stat_2dim_BYTE[k,l] := 1;
		stat_2dim_WORD[k,l] := 1;
		stat_2dim_DWORD[k,l] := 1;
		stat_2dim_LWORD[k,l] := 1;
		stat_2dim_R4[k,l] := 1.0;
		stat_2dim_R8[k,l] := 1.0;
		stat_2dim_BSTR[k,l] := 'Hello World';
		stat_2dim_WSTRING[k,l] := "Hello World";
		stat_2dim_DT[k,l] := DT#1972-03-29-00:00:00;
		stat_2dim_DATE[k,l] := DATE#1972-03-29;
		stat_2dim_TOD[k,l] := TOD#12:00:00;
		stat_2dim_TIME[k,l] := T#1S;
	END_FOR
END_FOR	

FOR m:= 0 TO ARRSIZEY DO
	FOR l:= 0 TO ARRSIZEY DO
		FOR k:= 0 TO ARRSIZEX DO
			stat_3dim_BOOL[k,l,m] := TRUE;
			stat_3dim_I1[k,l,m] := 1;
			stat_3dim_UI1[k,l,m] := 1;
			stat_3dim_I2[k,l,m] := 1;
			stat_3dim_UI2[k,l,m] := 1;
			stat_3dim_I4[k,l,m] := 1;
			stat_3dim_UI4[k,l,m] := 1;
			stat_3dim_I8[k,l,m] := 1;
			stat_3dim_UI8[k,l,m] := 1;
			stat_3dim_BYTE[k,l,m] := 1;
			stat_3dim_WORD[k,l,m] := 1;
			stat_3dim_DWORD[k,l,m] := 1;
			stat_3dim_LWORD[k,l,m] := 1;
			stat_3dim_R4[k,l,m] := 1.0;
			stat_3dim_R8[k,l,m] := 1.0;
			stat_3dim_BSTR[k,l,m] := 'Hello World';
			stat_3dim_WSTRING[k,l,m] := "Hello World";
			stat_3dim_DT[k,l,m] := DT#1972-03-29-00:00:00;
			stat_3dim_DATE[k,l,m] := DATE#1972-03-29;
			stat_3dim_TOD[k,l,m] := TOD#12:00:00;
			stat_3dim_TIME[k,l,m] := T#1S;			
		END_FOR
	END_FOR
END_FOR

END_PROGRAM

// ---- POUs/Programs/PRG_Dynamic.TcPOU
(* This program cyclically sets new values for variables in GVL_nodes_dynamic. *)
PROGRAM PRG_Dynamic
VAR
	(* Variables required for "running text" in STRING and WSTRING variables *)
	nTextMode :INT := 0;	
	sWordsU : WSTRING :=  "Hello OpcUA. Greetings from BECKHOFF AUTOMATION GmbH";
	sWordsA : STRING :=  'Hello OpcUA. Greetings from BECKHOFF AUTOMATION GmbH';
	idxEndChar :INT := 0;
	idxStartChar :INT := 1;
	
	(* Counter variables required to iterate through arrays *)
	k: INT;
	l: INT;
	m: INT;
END_VAR

(* Generate new data when timer triggers *)
Settings.UpdateTimer(IN:=TRUE);
IF Settings.UpdateTimer.Q THEN
	Settings.UpdateTimer(IN:=FALSE);
	
	(* Generate data for running text depending on text mode *)
	CASE nTextMode OF
		0:		
			idxStartChar := 1;
			idxEndChar :=idxEndChar+1;
			IF( idxEndChar > LEN( sWordsA ))THEN
				idxEndChar := LEN( sWordsA );
				idxStartChar :=1;	
				nTextMode := 1;
			END_IF
		1:
			idxEndChar := LEN( sWordsA );
			idxStartChar := idxStartChar+1;
			IF( idxStartChar >= LEN( sWordsA ))THEN
				idxStartChar := 1;	
				idxEndChar := 0	;		
				nTextMode := 0;
			END_IF
	END_CASE	
	
	(* Update scalar variables with new values *)
	GVL_nodes_dynamic.dyn_scalar_BOOL := NOT GVL_nodes_dynamic.dyn_scalar_BOOL;
	GVL_nodes_dynamic.dyn_scalar_I1 := GVL_nodes_dynamic.dyn_scalar_I1 + 1;
	GVL_nodes_dynamic.dyn_scalar_UI1 := GVL_nodes_dynamic.dyn_scalar_UI1 + 1;
	GVL_nodes_dynamic.dyn_scalar_I2	:= GVL_nodes_dynamic.dyn_scalar_I2 + 1;
	GVL_nodes_dynamic.dyn_scalar_UI2 := GVL_nodes_dynamic.dyn_scalar_UI2 + 1;
	GVL_nodes_dynamic.dyn_scalar_I4	:= GVL_nodes_dynamic.dyn_scalar_I4 + 1;
	GVL_nodes_dynamic.dyn_scalar_UI4 := GVL_nodes_dynamic.dyn_scalar_UI4 + 1;
	GVL_nodes_dynamic.dyn_scalar_I8	:= GVL_nodes_dynamic.dyn_scalar_I8  + 1;
	GVL_nodes_dynamic.dyn_scalar_UI8 := GVL_nodes_dynamic.dyn_scalar_UI8 + 1;
	GVL_nodes_dynamic.dyn_scalar_BYTE := GVL_nodes_dynamic.dyn_scalar_BYTE + 1;
	GVL_nodes_dynamic.dyn_scalar_WORD := GVL_nodes_dynamic.dyn_scalar_WORD + 1;
	GVL_nodes_dynamic.dyn_scalar_DWORD := GVL_nodes_dynamic.dyn_scalar_DWORD + 1;
	GVL_nodes_dynamic.dyn_scalar_LWORD := GVL_nodes_dynamic.dyn_scalar_LWORD + 1;
	GVL_nodes_dynamic.dyn_scalar_R4 := GVL_nodes_dynamic.dyn_scalar_R4 + 0.1;
	GVL_nodes_dynamic.dyn_scalar_R8 := GVL_nodes_dynamic.dyn_scalar_R8 + 0.1;
	GVL_nodes_dynamic.dyn_scalar_BSTR := MID(STR:=sWordsA, POS:=idxStartChar, LEN:=idxEndChar);
	GVL_nodes_dynamic.dyn_scalar_WSTRING := WMID(STR:=sWordsU, POS:=idxStartChar, LEN:=idxEndChar);
	GVL_nodes_dynamic.dyn_scalar_DT	:= GVL_nodes_dynamic.dyn_scalar_DT + T#1S;
	GVL_nodes_dynamic.dyn_scalar_DATE := GVL_nodes_dynamic.dyn_scalar_DATE + T#1S;
	GVL_nodes_dynamic.dyn_scalar_TOD := GVL_nodes_dynamic.dyn_scalar_TOD + T#1S;
	GVL_nodes_dynamic.dyn_scalar_TIME := GVL_nodes_dynamic.dyn_scalar_TIME + T#1S;
	
	(* Update array elements with new values *)
	FOR k:= 0 TO ARRSIZEHUGE DO
		GVL_nodes_dynamic.dyn_1dim_I1_Huge[k] := GVL_nodes_dynamic.dyn_1dim_I1_Huge[k]  +1;
		GVL_nodes_dynamic.dyn_1dim_I4_Huge[k] := GVL_nodes_dynamic.dyn_1dim_I4_Huge[k]  +1;
	END_FOR
	
	(* Update array elements with new values *)
	FOR k:= 0 TO ARRSIZEX DO
		GVL_nodes_dynamic.dyn_1dim_BOOL[k] := NOT GVL_nodes_dynamic.dyn_1dim_BOOL[k];
		GVL_nodes_dynamic.dyn_1dim_I1[k] := GVL_nodes_dynamic.dyn_1dim_I1[k] + 1;
		GVL_nodes_dynamic.dyn_1dim_UI1[k] := GVL_nodes_dynamic.dyn_1dim_UI1[k] + 1;
		GVL_nodes_dynamic.dyn_1dim_I2[k] := GVL_nodes_dynamic.dyn_1dim_I2[k] + 1;
		GVL_nodes_dynamic.dyn_1dim_UI2[k] := GVL_nodes_dynamic.dyn_1dim_UI2[k] + 1;
		GVL_nodes_dynamic.dyn_1dim_I4[k] := GVL_nodes_dynamic.dyn_1dim_I4[k] + 1;
		GVL_nodes_dynamic.dyn_1dim_UI4[k] := GVL_nodes_dynamic.dyn_1dim_UI4[k] + 1;
		GVL_nodes_dynamic.dyn_1dim_I8[k] := GVL_nodes_dynamic.dyn_1dim_I8[k] + 1;
		GVL_nodes_dynamic.dyn_1dim_UI8[k] := GVL_nodes_dynamic.dyn_1dim_UI8[k] + 1;
		GVL_nodes_dynamic.dyn_1dim_BYTE[k] := GVL_nodes_dynamic.dyn_1dim_BYTE[k] + 1;
		GVL_nodes_dynamic.dyn_1dim_WORD[k] := GVL_nodes_dynamic.dyn_1dim_WORD[k] + 1;
		GVL_nodes_dynamic.dyn_1dim_DWORD[k] := GVL_nodes_dynamic.dyn_1dim_DWORD[k] + 1;
		GVL_nodes_dynamic.dyn_1dim_LWORD[k] := GVL_nodes_dynamic.dyn_1dim_LWORD[k] + 1;
		GVL_nodes_dynamic.dyn_1dim_R4[k] := GVL_nodes_dynamic.dyn_1dim_R4[k] + 0.1;
		GVL_nodes_dynamic.dyn_1dim_R8[k] := GVL_nodes_dynamic.dyn_1dim_R8[k] + 0.1;
		GVL_nodes_dynamic.dyn_1dim_BSTR[k] := MID(STR:=sWordsA, POS:=idxStartChar, LEN:=idxEndChar);
		GVL_nodes_dynamic.dyn_1dim_WSTRING[k] := WMID(STR:=sWordsU, POS:=idxStartChar, LEN:=idxEndChar);
		GVL_nodes_dynamic.dyn_1dim_DT[k] := GVL_nodes_dynamic.dyn_1dim_DT[k] + T#1S;
		GVL_nodes_dynamic.dyn_1dim_DATE[k] := GVL_nodes_dynamic.dyn_1dim_DATE[k] + T#1S;
		GVL_nodes_dynamic.dyn_1dim_TOD[k] := GVL_nodes_dynamic.dyn_1dim_TOD[k] + T#1S;
		GVL_nodes_dynamic.dyn_1dim_TIME[k] := GVL_nodes_dynamic.dyn_1dim_TIME[k] + T#1S;
	END_FOR;
	
	(* Update 2-dim array elements with new values *)
	FOR l:= 0 TO ARRSIZEY DO
		FOR k:= 0 TO ARRSIZEX DO
			GVL_nodes_dynamic.dyn_2dim_BOOL[k,l] := NOT GVL_nodes_dynamic.dyn_2dim_BOOL[k,l];
			GVL_nodes_dynamic.dyn_2dim_I1[k,l] := GVL_nodes_dynamic.dyn_2dim_I1[k,l] + 1;
			GVL_nodes_dynamic.dyn_2dim_UI1[k,l] := GVL_nodes_dynamic.dyn_2dim_UI1[k,l] + 1;
			GVL_nodes_dynamic.dyn_2dim_I2[k,l] := GVL_nodes_dynamic.dyn_2dim_I2[k,l] + 1;
			GVL_nodes_dynamic.dyn_2dim_UI2[k,l] := GVL_nodes_dynamic.dyn_2dim_UI2[k,l] + 1;
			GVL_nodes_dynamic.dyn_2dim_I4[k,l] := GVL_nodes_dynamic.dyn_2dim_I4[k,l] + 1;
			GVL_nodes_dynamic.dyn_2dim_UI4[k,l] := GVL_nodes_dynamic.dyn_2dim_UI4[k,l] + 1;
			GVL_nodes_dynamic.dyn_2dim_I8[k,l] := GVL_nodes_dynamic.dyn_2dim_I8[k,l] + 1;
			GVL_nodes_dynamic.dyn_2dim_UI8[k,l] := GVL_nodes_dynamic.dyn_2dim_UI8[k,l] + 1;
			GVL_nodes_dynamic.dyn_2dim_BYTE[k,l] := GVL_nodes_dynamic.dyn_2dim_BYTE[k,l] + 1;
			GVL_nodes_dynamic.dyn_2dim_WORD[k,l] := GVL_nodes_dynamic.dyn_2dim_WORD[k,l] + 1;
			GVL_nodes_dynamic.dyn_2dim_DWORD[k,l] := GVL_nodes_dynamic.dyn_2dim_DWORD[k,l] + 1;
			GVL_nodes_dynamic.dyn_2dim_LWORD[k,l] := GVL_nodes_dynamic.dyn_2dim_LWORD[k,l] + 1;
			GVL_nodes_dynamic.dyn_2dim_R4[k,l] := GVL_nodes_dynamic.dyn_2dim_R4[k,l] + 0.1;
			GVL_nodes_dynamic.dyn_2dim_R8[k,l] := GVL_nodes_dynamic.dyn_2dim_R8[k,l] + 0.1;
			GVL_nodes_dynamic.dyn_2dim_BSTR[k,l] := MID(STR:=sWordsA, POS:=idxStartChar, LEN:=idxEndChar);
			GVL_nodes_dynamic.dyn_2dim_WSTRING[k,l] := WMID(STR:=sWordsU, POS:=idxStartChar, LEN:=idxEndChar);
			GVL_nodes_dynamic.dyn_2dim_DT[k,l] := GVL_nodes_dynamic.dyn_2dim_DT[k,l] + T#1S;
			GVL_nodes_dynamic.dyn_2dim_DATE[k,l] := GVL_nodes_dynamic.dyn_2dim_DATE[k,l] + T#1S;
			GVL_nodes_dynamic.dyn_2dim_TOD[k,l] := GVL_nodes_dynamic.dyn_2dim_TOD[k,l] + T#1S;
			GVL_nodes_dynamic.dyn_2dim_TIME[k,l] := GVL_nodes_dynamic.dyn_2dim_TIME[k,l] + T#1S;
		END_FOR;
	END_FOR;
	
	(* Update 3-dim array elements with new values *)
	FOR m:= 0 TO ARRSIZEY DO
		FOR l:= 0 TO ARRSIZEY DO
			FOR k:= 0 TO ARRSIZEX DO
				GVL_nodes_dynamic.dyn_3dim_BOOL[k,l,m] := NOT GVL_nodes_dynamic.dyn_3dim_BOOL[k,l,m];
				GVL_nodes_dynamic.dyn_3dim_I1[k,l,m] := GVL_nodes_dynamic.dyn_3dim_I1[k,l,m] + 1;
				GVL_nodes_dynamic.dyn_3dim_UI1[k,l,m] := GVL_nodes_dynamic.dyn_3dim_UI1[k,l,m] + 1;
				GVL_nodes_dynamic.dyn_3dim_I2[k,l,m] := GVL_nodes_dynamic.dyn_3dim_I2[k,l,m] + 1;
				GVL_nodes_dynamic.dyn_3dim_UI2[k,l,m] := GVL_nodes_dynamic.dyn_3dim_UI2[k,l,m] + 1;
				GVL_nodes_dynamic.dyn_3dim_I4[k,l,m] := GVL_nodes_dynamic.dyn_3dim_I4[k,l,m] + 1;
				GVL_nodes_dynamic.dyn_3dim_UI4[k,l,m] := GVL_nodes_dynamic.dyn_3dim_UI4[k,l,m] + 1;
				GVL_nodes_dynamic.dyn_3dim_I8[k,l,m] := GVL_nodes_dynamic.dyn_3dim_I8[k,l,m] + 1;
				GVL_nodes_dynamic.dyn_3dim_UI8[k,l,m] := GVL_nodes_dynamic.dyn_3dim_UI8[k,l,m] + 1;
				GVL_nodes_dynamic.dyn_3dim_BYTE[k,l,m] := GVL_nodes_dynamic.dyn_3dim_BYTE[k,l,m] + 1;
				GVL_nodes_dynamic.dyn_3dim_WORD[k,l,m] := GVL_nodes_dynamic.dyn_3dim_WORD[k,l,m] + 1;
				GVL_nodes_dynamic.dyn_3dim_DWORD[k,l,m] := GVL_nodes_dynamic.dyn_3dim_DWORD[k,l,m] + 1;
				GVL_nodes_dynamic.dyn_3dim_LWORD[k,l,m] := GVL_nodes_dynamic.dyn_3dim_LWORD[k,l,m] + 1;
				GVL_nodes_dynamic.dyn_3dim_R4[k,l,m] := GVL_nodes_dynamic.dyn_3dim_R4[k,l,m] + 0.1;
				GVL_nodes_dynamic.dyn_3dim_R8[k,l,m] := GVL_nodes_dynamic.dyn_3dim_R8[k,l,m] + 0.1;
				GVL_nodes_dynamic.dyn_3dim_BSTR[k,l,m] := MID(STR:=sWordsA, POS:=idxStartChar, LEN:=idxEndChar);
				GVL_nodes_dynamic.dyn_3dim_WSTRING[k,l,m] := WMID(STR:=sWordsU, POS:=idxStartChar, LEN:=idxEndChar);
				GVL_nodes_dynamic.dyn_3dim_DT[k,l,m] := GVL_nodes_dynamic.dyn_3dim_DT[k,l,m] + T#1S;
				GVL_nodes_dynamic.dyn_3dim_DATE[k,l,m] := GVL_nodes_dynamic.dyn_3dim_DATE[k,l,m] + T#1S;
				GVL_nodes_dynamic.dyn_3dim_TOD[k,l,m] := GVL_nodes_dynamic.dyn_3dim_TOD[k,l,m] + T#1S;
				GVL_nodes_dynamic.dyn_3dim_TIME[k,l,m] := GVL_nodes_dynamic.dyn_3dim_TIME[k,l,m] + T#1S;
			END_FOR;
		END_FOR;
	END_FOR;
END_IF

END_PROGRAM

// ---- POUs/Programs/PRG_Eventlogger.TcPOU
(* This program is based on the standard TcEventlogger sample and provides sample code to fire an alarm and event
   The TcOpcUaServer can be configured to subscribe to TcEventlogger alarms and events and convert them into an 
   OPC UA alarm/event. Please consult the TF6100 documentation on the Beckhoff Information System fore more info *) 
PROGRAM PRG_Eventlogger
VAR
	bInit : BOOL := TRUE; 
    bSend : BOOL := FALSE;	
	bAlmRaise : BOOL := FALSE;
	bAlmConfirm : BOOL := FALSE;
	bAlmClear : BOOL := FALSE;
    fbMsg : FB_TcMessage;
	fbAlm : FB_TcAlarm; 	
END_VAR

IF bInit THEN
    bInit := FALSE; 
    fbMsg.CreateEx(TC_EVENTS.TutorialClass.Event, 0); 
	fbAlm.CreateEx(TC_EVENTS.TutorialClass.Alarm, TRUE, 0, );
END_IF

IF bSend THEN 
    bSend := FALSE;
	fbMsg.SetJsonAttribute( '{"name":"fbMsg", "action":"send"}' );
    fbMsg.Send(0); 
END_IF

IF bAlmRaise THEN
	bAlmRaise := FALSE;
	fbAlm.SetJsonAttribute( '{"name":"fbAlm", "action":"Raise"}' );
	fbAlm.Raise(0);
END_IF

IF bAlmConfirm THEN
	bAlmConfirm := FALSE;
	fbAlm.SetJsonAttribute( '{"name":"fbAlm", "action":"Confirm"}' );
	fbAlm.Confirm(0);
END_IF
	
IF bAlmClear THEN
	bAlmClear := FALSE;
	fbAlm.SetJsonAttribute( '{"name":"fbAlm", "action":"Clear"}' );
	fbAlm.Clear(0, FALSE);
END_IF

END_PROGRAM

// ---- POUs/Programs/PRG_HistoricalAccess.TcPOU
(* Generates data for variables in GVL_historizing, which are used by server for Historical Access. *)
PROGRAM PRG_HistoricalAccess
VAR
	i : INT;
	o : LREAL;
	Sinus : LREAL;
	Cosinus : LREAL;
	Cosinus_Half : LREAL;
	Ts : INT;	
END_VAR

i := i + 1;
o := o + 0.001;
Ts := 128 * 10;

Sinus := SIN(o);
Cosinus := COS(o);
Cosinus_Half:=COS(PI * i / (2 * Ts));

(* Update global variables in GVL_historizing, which are being used by server for HA *)
GVL_historizing.volatile_sinus := Sinus;  
GVL_historizing.volatile_cosinus := Cosinus;
GVL_historizing.volatile_cosinushalf := Cosinus_Half;  

GVL_historizing.sqlite_sinus := Sinus;
GVL_historizing.sqlite_cosinus := Cosinus;
GVL_historizing.sqlite_cosinushalf := Cosinus_Half;

END_PROGRAM

// ---- POUs/Programs/PRG_AlarmsConditions.TcPOU
PROGRAM PRG_AlarmsConditions
VAR
	(* HiHi and LoLo values for variable to trigger LimitAlarmType *)
	nLimitAlarmTypeUpperLimit : INT := 10;
	nLimitAlarmTypeLowerLimit : INT := 0;
    bCountUp : BOOL := TRUE;

	(* Timer variables *)
	timer_1s : TON := (PT:=T#1S); // used for LimitAlarmType
	timer_10s : TON := (PT:=T#10S); // used for OffNormalAlarmType
END_VAR

(* Execute when timer triggers *)
timer_1s(IN := TRUE);
IF( timer_1s.Q ) THEN
	timer_1s( in:=FALSE );
	// Generate a cyclic up/down ramp for the limit alarm trigger value.
	// The value is incremented until the upper limit is reached.
	// Afterwards, the direction is changed and the value is decremented
	// until the lower limit is reached. The bCountUp flag stores the
	// current counting direction.
	IF bCountUp THEN
		GVL_alarm_condition.limitAlmTrigger := GVL_alarm_condition.limitAlmTrigger + 1;
		IF GVL_alarm_condition.limitAlmTrigger >= nLimitAlarmTypeUpperLimit THEN
			GVL_alarm_condition.limitAlmTrigger := nLimitAlarmTypeUpperLimit;
			bCountUp := FALSE;
		END_IF
	ELSE
		GVL_alarm_condition.limitAlmTrigger := GVL_alarm_condition.limitAlmTrigger - 1;
		IF GVL_alarm_condition.limitAlmTrigger <= nLimitAlarmTypeLowerLimit THEN
			GVL_alarm_condition.limitAlmTrigger := nLimitAlarmTypeLowerLimit;
			bCountUp := TRUE;
		END_IF
	END_IF	
END_IF

(* Execute when timer triggers *)
timer_10s(IN := TRUE);
IF( timer_10s.Q ) THEN
	timer_10s( in:=FALSE );
	// Generate a cyclic Boolean trigger value for the OffNormal alarm.
	// The value is toggled whenever the timer elapses, causing the
	// OffNormal alarm condition to periodically become active and inactive.
	GVL_alarm_condition.offNormAlmTrigger := NOT GVL_alarm_condition.offNormAlmTrigger;
END_IF

END_PROGRAM

// ---- POUs/Programs/PRG_Methods.TcPOU
PROGRAM PRG_Methods
VAR
END_VAR

GVL_methods.Job(); // Cyclic execution of function block that is exposed as "job method"

END_PROGRAM

// ---- POUs/Inheritance/FB_Base.TcPOU
FUNCTION_BLOCK FB_Base
VAR_INPUT
	Input1 : INT;
	Input2 : REAL;
END_VAR
VAR_OUTPUT
	Output1 : DINT;
	Output2 : LREAL;
END_VAR
VAR
	Internal1 : SINT;
	Internal2 : WORD;
	Internal3 : ST_Complex_1;
END_VAR

END_FUNCTION_BLOCK

// ---- POUs/Inheritance/FB_Derived.TcPOU
FUNCTION_BLOCK FB_Derived EXTENDS FB_Base
VAR_INPUT
	DerivedInput1 : INT;
	DerivedInput2 : REAL;
END_VAR
VAR_OUTPUT
	DerivedOutput1 : DINT;
	DerivedOutput2 : LREAL;
END_VAR
VAR
	DerivedInternal1 : SINT;
	DerivedInternal2 : WORD;
END_VAR

END_FUNCTION_BLOCK

// ---- POUs/Properties/FB_Properties.TcPOU
FUNCTION_BLOCK FB_Properties
VAR_INPUT
END_VAR
VAR_OUTPUT
END_VAR
VAR
END_VAR

{attribute 'OPC.UA.DA.Property' := '1'}
{attribute 'monitoring' := 'call'}
PROPERTY MyProperty1 : BOOL
GET
END_GET
SET
END_SET
END_PROPERTY

END_FUNCTION_BLOCK

// ---- POUs/Methods/FB_Methods.TcPOU
FUNCTION_BLOCK FB_Methods
VAR
	count : LREAL;
END_VAR

{attribute 'TcRpcEnable'}
{attribute 'OPC.UA.DA.Description' := 'Returns array of INT'}
METHOD M_Array_1 : ARRAY[0..2] OF INT
VAR_INPUT
END_VAR
VAR
	aTest : ARRAY[0..2] OF INT;
END_VAR
aTest[0] := 1;
aTest[1] := 2;
aTest[2] := 3;
M_Array_1 := aTest;
END_METHOD

{attribute 'TcRpcEnable'}
{attribute 'OPC.UA.DA.Description' := 'Returns array of INT'}
METHOD M_Array_2 : ARRAY[0..9] OF INT
VAR_INPUT
	aTest : ARRAY[0..9] OF INT;
END_VAR
M_Array_2 := aTest;
END_METHOD

{attribute 'TcRpcEnable'}
{attribute 'OPC.UA.DA.Description' := 'Returns simple complex type'}
METHOD M_Complex_1 : ST_Complex_1
count :=count+1;
M_Complex_1.a := 1;
M_Complex_1.b := 2;
END_METHOD

{attribute 'TcRpcEnable'}
{attribute 'OPC.UA.DA.Description' := 'InOut argument is a simple complex type'}
METHOD M_Complex_2 : ST_Complex_1
VAR_INPUT
	in : ST_Complex_1;
END_VAR
count :=count+1;
M_Complex_2.a := in.a + 1;
M_Complex_2.b := in.b + 1;
END_METHOD

{attribute 'TcRpcEnable'}
{attribute 'OPC.UA.DA.Description' := 'Method without InOut arguments'}
METHOD M_NoArgs
VAR_INPUT
END_VAR
count :=count+1;
END_METHOD

END_FUNCTION_BLOCK

// ---- POUs/Methods/FB_Mathematics.TcPOU
FUNCTION_BLOCK FB_Mathematics
VAR
	count : LREAL;
END_VAR

{attribute 'TcRpcEnable'}
{attribute 'OPC.UA.DA.Description' := 'Returns a + b'}
METHOD Add2 : LREAL
VAR_INPUT
	a : LREAL;(*Value 'a'*)
	b : LREAL; (*Value 'b'*)
END_VAR
count :=count+1;
Add2 := a+b;
END_METHOD

{attribute 'TcRpcEnable'}
{attribute 'OPC.UA.DA.Description' := 'Perform calculation on a and b, as defined by value operation'}
METHOD Calculate : LREAL
VAR_INPUT	
	operation : E_OPERATION; (*define the kind of operation to be done*)
	a : LREAL; (*Value for a*)
	b: LREAL; (*Value for b*)
END_VAR
count :=count+1;
Calculate := 0;
CASE operation OF
	Addition:
		Calculate := a+b;
	Substract:
		Calculate := a-b;
	Multiply:
		Calculate := a*b;
	Divide:
		Calculate := a/b;	
END_CASE
END_METHOD

{attribute 'TcRpcEnable'}
{attribute 'OPC.UA.DA.Description' := 'Perform calculation as described in Parameter o'}
METHOD Calculate2 : LREAL
VAR_INPUT
	in : ST_MathOperation; (*structure, defining the calculation to be done*)
END_VAR
count :=count+1;
CASE in.operator OF
	Addition:
		Calculate2 := in.a+in.b;
	Substract:
		Calculate2 := in.a-in.b;
	Multiply:
		Calculate2 := in.a*in.b;
	Divide:
		Calculate2 := in.a/in.b;
END_CASE
END_METHOD

{attribute 'TcRpcEnable'}
{attribute 'OPC.UA.DA.Description' := 'Perform calculation and return results as STRING'}
METHOD Calculate3 : STRING
VAR_INPUT
	operation : E_OPERATION; (*define the kind of operation to be done*)
	a:INT;
	b:INT;
END_VAR
count :=count+1;
CASE operation OF
	Addition:
		Calculate3 := DINT_TO_STRING(a+b);
	Substract:
		Calculate3 := DINT_TO_STRING(a-b);
	Multiply:
		Calculate3 := DINT_TO_STRING(a*b);
	Divide:
		Calculate3 := DINT_TO_STRING(a/b);	
END_CASE
END_METHOD

{attribute 'TcRpcEnable'}
{attribute 'OPC.UA.DA.Description' := 'Perform calculation and return results as STRING'}
METHOD Calculate4 : STRING
VAR_INPUT
	a:INT;
	b:INT;
END_VAR
VAR_OUTPUT
	sMul: STRING;
	sSub: STRING;
END_VAR
count :=count+1;
Calculate4 := DINT_TO_STRING(a + b);
sMul := DINT_TO_STRING(a * b);
sSub := INT_TO_STRING(a - b);
END_METHOD

{attribute 'TcRpcEnable'}
{attribute 'OPC.UA.DA.Description' := 'Perform calculation and return results as STRING'}
METHOD Calculate5 : ST_MathematicResults
VAR_INPUT
	a:INT;
	b:INT;
END_VAR
count :=count+1;
Calculate5.Diff := a - b;
Calculate5.Prod := a * b;
Calculate5.Quo := a / b;
Calculate5.Sum := a + b;
END_METHOD

{attribute 'TcRpcEnable'} 
METHOD Div2 : LREAL
VAR_INPUT
	a:LREAL;
	b:LREAL;
END_VAR
count :=count+1;
Div2 := a/b;
END_METHOD

{attribute 'TcRpcEnable'} 
METHOD Mul2 : LREAL
VAR_INPUT
	a:LREAL;
	b:LREAL;
END_VAR
count :=count+1;
Mul2:= a*b;
END_METHOD

{attribute 'TcRpcEnable'} 
METHOD Sub2 : LREAL
VAR_INPUT
	a:LREAL;
	b:LREAL;
END_VAR
count :=count+1;
Sub2:=a-b;
END_METHOD

END_FUNCTION_BLOCK

// ---- POUs/Methods/FB_Job.TcPOU
{attribute 'OPC.UA.DA.JobMethod' := 'MyJob'}
FUNCTION_BLOCK FB_Job
VAR
	// Used for debugging purposes to display InputArguments of method call
	Input_a : INT; // used to store InputArg "a" from Start() method
	Input_b : LREAL; // used to store InputArg "b" from Start() method
	Input_c : BOOL; // used to store InputArg "c" from Start() method
	Input_d : ST_Complex_1; // used to store InputArg "d" from Start() method
	callCounterStart : ULINT; // counts how many times the Start() method has been called
	callCounterCheckState : ULINT; // counts how many times the CheckState() method has been called
	callCounterAbort : ULINT; // counts how many times the Abort() method has been called
	
	// Timer to "artificially delay" job execution
	timer : TON := (PT:=T#4S);
	
	// Variables to determine if a job has been started (Start() method has been called) or finished
	jobRunning : BOOL;
	jobFinished : BOOL;

	// State machine variable
	state : UDINT;
END_VAR

CASE state OF
	0:
		IF jobRunning THEN
			state := state + 1;
		END_IF
		
	1:
		timer(IN:=TRUE);
		IF timer.Q THEN
			timer(IN:=FALSE);
			jobRunning := FALSE;
			jobFinished := TRUE;
			state := 0;
		END_IF
		
END_CASE

{attribute 'TcRpcEnable' := '1'}
METHOD Abort : HRESULT
VAR_INPUT
	hdl : UDINT; // Do not change, used by server.
END_VAR
callCounterAbort := callCounterAbort + 1;
END_METHOD

{attribute 'TcRpcEnable' := '1'}
METHOD CheckState : HRESULT
VAR_INPUT
	hdl : UDINT; // Do not change, used by server.
END_VAR
VAR_OUTPUT
	bBusy : BOOL; // Do not change. Used by server to find out if the job is finished
	
	// List of OutputArguments for OPC UA method, may be customized
	a : INT; // some description
	b : LREAL; // some description
	c : BOOL; // some description
	d : ST_Complex_1; // some description
END_VAR
callCounterCheckState := callCounterCheckState + 1;
IF NOT jobFinished THEN
	bBusy := TRUE; // job is not finished yet
	CheckState := 0; // no error
ELSE
	bBusy := FALSE; // job is finished
	CheckState := 0; // done, no error occured during execution (OPC UA StatusCode "GOOD")
	jobFinished := FALSE;
	a := Input_a;
	b := Input_b;
	c := Input_c;
	d := Input_d;
END_IF
END_METHOD

{attribute 'TcRpcEnable' := '1'}
METHOD Start : HRESULT
VAR_INPUT
	// List of InputArguments for OPC UA method, may be customized
	a : INT; // some description
	b : LREAL; // some description
	c : BOOL; // some description
	d : ST_Complex_1; // some description
END_VAR
VAR_OUTPUT
	hdl : UDINT; // Do not change, used by server.
END_VAR
callCounterStart := callCounterStart + 1;
Input_a := a;
Input_b := b;
Input_c := c;
Input_d := d;
jobRunning := TRUE;
Start := 0; // no error occured, e.g. while parsing the input arguments (0 = OPC UA StatusCode "GOOD")
END_METHOD

END_FUNCTION_BLOCK
